KUKA KRL program: MyProgram_004().src

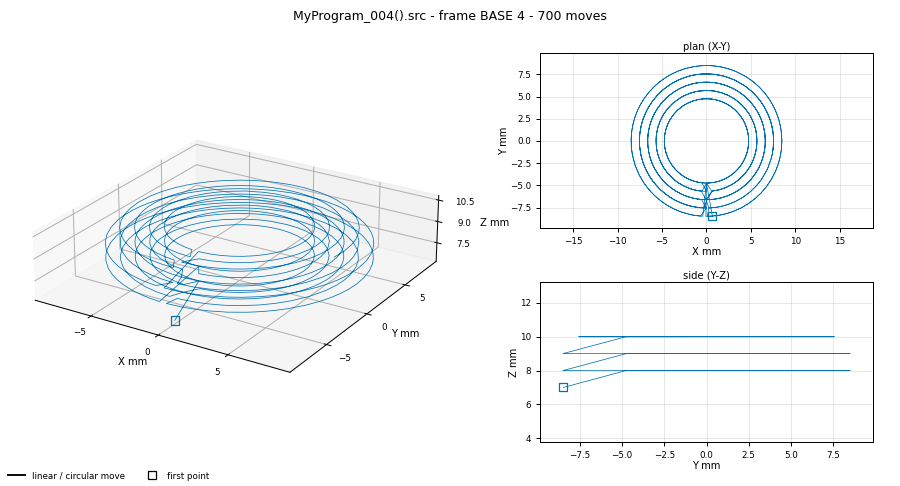
[picture p0: tool path of MyProgram_004().src in frame BASE 4, 700 of 700 moves have a stored position in this frame; points joined in program order, loops and branches not executed]
&ACCESS RVP
&REL 1
&PARAM TEMPLATE = C:\KRC\Roboter\Template\vorgabe
&PARAM EDITMASK = *
DEF MyProgram_004()
; ---- Setting reference (Base) ----
$BASE = BASE_DATA[4]

; --------------------------
; ---- Setting tool (TCP) ----
$TOOL = TOOL_DATA[3]
; --------------------------

$VEL.CP = VEL_APROX_PRINT
Startdeposition()
$VEL.CP = VEL_PRINT
LIN {X 0.6654,Y -8.462,Z 7,A -3.1447,B 0,C 0,E1 0.1598,E2 90.0714} C_DIS
Enddeposition()
LIN {X 0.0002,Y -4.7529,Z 8,A -2.9966,B 0,C 0,E1 0.1598,E2 90.0603} C_DIS
Startdeposition()
$VEL.CP = VEL_PRINT
LIN {X 0.0002,Y -4.7529,Z 8,A -3.0023,B 0,C 0,E1 0.1598,E2 90.066} C_DIS
LIN {X 0.816,Y -4.6799,Z 8,A -2.9741,B 0,C 0,E1 0.1598,E2 90.0709} C_DIS
LIN {X 1.4524,Y -4.5228,Z 8,A -2.9447,B 0,C 0,E1 0.1598,E2 90.0716} C_DIS
LIN {X 2.0618,Y -4.2811,Z 8,A -2.9121,B 0,C 0,E1 0.1598,E2 90.0716} C_DIS
LIN {X 2.6304,Y -3.9547,Z 8,A -2.8774,B 0,C 0,E1 0.1598,E2 90.0716} C_DIS
LIN {X 3.1509,Y -3.5562,Z 8,A -2.8413,B 0,C 0,E1 0.1598,E2 90.0717} C_DIS
LIN {X 3.6101,Y -3.0885,Z 8,A -2.8046,B 0,C 0,E1 0.1598,E2 90.0717} C_DIS
LIN {X 4.0002,Y -2.5617,Z 8,A -2.7679,B 0,C 0,E1 0.1598,E2 90.0717} C_DIS
LIN {X 4.3166,Y -1.9875,Z 8,A -2.7319,B 0,C 0,E1 0.1598,E2 90.0717} C_DIS
LIN {X 4.5475,Y -1.3739,Z 8,A -2.6974,B 0,C 0,E1 0.1598,E2 90.0717} C_DIS
LIN {X 4.6933,Y -0.7348,Z 8,A -2.6649,B 0,C 0,E1 0.1598,E2 90.0718} C_DIS
LIN {X 4.7495,Y -0.0819,Z 8,A -2.6352,B 0,C 0,E1 0.1598,E2 90.0718} C_DIS
LIN {X 4.7181,Y 0.573,Z 8,A -2.6086,B 0,C 0,E1 0.1598,E2 90.0718} C_DIS
LIN {X 4.5916,Y 1.2163,Z 8,A -2.586,B 0,C 0,E1 0.1598,E2 90.0718} C_DIS
LIN {X 4.3818,Y 1.8374,Z 8,A -2.5674,B 0,C 0,E1 0.1598,E2 90.0719} C_DIS
LIN {X 4.0877,Y 2.4234,Z 8,A -2.5534,B 0,C 0,E1 0.1598,E2 90.0719} C_DIS
LIN {X 3.7147,Y 2.9626,Z 8,A -2.5444,B 0,C 0,E1 0.1598,E2 90.072} C_DIS
LIN {X 3.2724,Y 3.4466,Z 8,A -2.5402,B 0,C 0,E1 0.1598,E2 90.072} C_DIS
LIN {X 2.7665,Y 3.864,Z 8,A -2.5413,B 0,C 0,E1 0.1598,E2 90.072} C_DIS
LIN {X 2.2075,Y 4.2066,Z 8,A -2.5474,B 0,C 0,E1 0.1598,E2 90.0721} C_DIS
LIN {X 1.6077,Y 4.4708,Z 8,A -2.5584,B 0,C 0,E1 0.1598,E2 90.0721} C_DIS
LIN {X 0.977,Y 4.6499,Z 8,A -2.5741,B 0,C 0,E1 0.1598,E2 90.0721} C_DIS
LIN {X 0.3277,Y 4.7412,Z 8,A -2.5942,B 0,C 0,E1 0.1598,E2 90.0721} C_DIS
LIN {X -0.3279,Y 4.7398,Z 8,A -2.6184,B 0,C 0,E1 0.1598,E2 90.0721} C_DIS
LIN {X -0.977,Y 4.6484,Z 8,A -2.6462,B 0,C 0,E1 0.1598,E2 90.0721} C_DIS
LIN {X -1.608,Y 4.4707,Z 8,A -2.677,B 0,C 0,E1 0.1598,E2 90.072} C_DIS
LIN {X -2.2078,Y 4.2061,Z 8,A -2.7102,B 0,C 0,E1 0.1598,E2 90.072} C_DIS
LIN {X -2.766,Y 3.862,Z 8,A -2.7453,B 0,C 0,E1 0.1598,E2 90.0719} C_DIS
LIN {X -3.2729,Y 3.4465,Z 8,A -2.7815,B 0,C 0,E1 0.1598,E2 90.0718} C_DIS
LIN {X -3.715,Y 2.9623,Z 8,A -2.8181,B 0,C 0,E1 0.1598,E2 90.0718} C_DIS
LIN {X -4.0878,Y 2.4229,Z 8,A -2.8545,B 0,C 0,E1 0.1598,E2 90.0716} C_DIS
LIN {X -4.3815,Y 1.8369,Z 8,A -2.89,B 0,C 0,E1 0.1598,E2 90.0716} C_DIS
LIN {X -4.5933,Y 1.2164,Z 8,A -2.924,B 0,C 0,E1 0.1598,E2 90.0715} C_DIS
LIN {X -4.7177,Y 0.5725,Z 8,A -2.9556,B 0,C 0,E1 0.1598,E2 90.0715} C_DIS
LIN {X -4.7506,Y -0.0822,Z 8,A -2.9844,B 0,C 0,E1 0.1598,E2 90.0714} C_DIS
LIN {X -4.6934,Y -0.7352,Z 8,A -3.0099,B 0,C 0,E1 0.1598,E2 90.0714} C_DIS
LIN {X -4.5474,Y -1.3743,Z 8,A -3.0314,B 0,C 0,E1 0.1598,E2 90.0714} C_DIS
LIN {X -4.3157,Y -1.9876,Z 8,A -3.0488,B 0,C 0,E1 0.1598,E2 90.0714} C_DIS
LIN {X -4.0017,Y -2.5632,Z 8,A -3.0616,B 0,C 0,E1 0.1598,E2 90.0714} C_DIS
LIN {X -3.6098,Y -3.0888,Z 8,A -3.0694,B 0,C 0,E1 0.1598,E2 90.0714} C_DIS
LIN {X -3.1503,Y -3.5561,Z 8,A -3.0722,B 0,C 0,E1 0.1598,E2 90.0714} C_DIS
LIN {X -2.6304,Y -3.9555,Z 8,A -3.0701,B 0,C 0,E1 0.1598,E2 90.0714} C_DIS
LIN {X -2.061,Y -4.2801,Z 8,A -3.0629,B 0,C 0,E1 0.1598,E2 90.0714} C_DIS
LIN {X -1.4527,Y -4.525,Z 8,A -3.0509,B 0,C 0,E1 0.1598,E2 90.0714} C_DIS
LIN {X -0.8159,Y -4.6817,Z 8,A -3.0342,B 0,C 0,E1 0.1598,E2 90.0715} C_DIS
LIN {X 0.0002,Y -4.7529,Z 8,A -3.0072,B 0,C 0,E1 0.1598,E2 90.0715} C_DIS
Enddeposition()
LIN {X 0.0002,Y -4.7529,Z 8,A -3.0072,B 0,C 0,E1 0.1598,E2 90.0715} C_DIS
Startdeposition()
$VEL.CP = VEL_PRINT
LIN {X -0.5157,Y -5.66,Z 8,A -3.0641,B 0,C 0,E1 0.1598,E2 90.0709} C_DIS
LIN {X -1.2329,Y -5.5494,Z 8,A -3.0863,B 0,C 0,E1 0.1598,E2 90.0714} C_DIS
LIN {X -2.1019,Y -5.2885,Z 8,A -3.1072,B 0,C 0,E1 0.1598,E2 90.0714} C_DIS
LIN {X -3.0914,Y -4.7699,Z 8,A -3.1214,B 0,C 0,E1 0.1598,E2 90.0712} C_DIS
LIN {X -3.7339,Y -4.2857,Z 8,A -3.1246,B 0,C 0,E1 0.1598,E2 90.0712} C_DIS
LIN {X -4.3031,Y -3.7167,Z 8,A -3.1215,B 0,C 0,E1 0.1598,E2 90.0712} C_DIS
LIN {X -4.784,Y -3.0715,Z 8,A -3.1119,B 0,C 0,E1 0.1598,E2 90.0712} C_DIS
LIN {X -5.0868,Y -2.5489,Z 8,A -3.101,B 0,C 0,E1 0.1598,E2 90.0713} C_DIS
LIN {X -5.4926,Y -1.467,Z 8,A -3.0698,B 0,C 0,E1 0.1598,E2 90.0708} C_DIS
LIN {X -5.6398,Y -0.761,Z 8,A -3.0457,B 0,C 0,E1 0.1598,E2 90.0711} C_DIS
LIN {X -5.6808,Y 0.176,Z 8,A -3.0077,B 0,C 0,E1 0.1598,E2 90.0711} C_DIS
LIN {X -5.6091,Y 0.9228,Z 8,A -2.9738,B 0,C 0,E1 0.1598,E2 90.0713} C_DIS
LIN {X -5.4394,Y 1.6537,Z 8,A -2.9367,B 0,C 0,E1 0.1598,E2 90.0713} C_DIS
LIN {X -5.1717,Y 2.3546,Z 8,A -2.8974,B 0,C 0,E1 0.1598,E2 90.0715} C_DIS
LIN {X -4.8184,Y 3.0165,Z 8,A -2.8565,B 0,C 0,E1 0.1598,E2 90.0715} C_DIS
LIN {X -4.3794,Y 3.6251,Z 8,A -2.8147,B 0,C 0,E1 0.1598,E2 90.0716} C_DIS
LIN {X -3.863,Y 4.1692,Z 8,A -2.7728,B 0,C 0,E1 0.1598,E2 90.0717} C_DIS
LIN {X -2.9369,Y 4.873,Z 8,A -2.7089,B 0,C 0,E1 0.1598,E2 90.0717} C_DIS
LIN {X -1.8956,Y 5.3645,Z 8,A -2.6499,B 0,C 0,E1 0.1598,E2 90.0719} C_DIS
LIN {X -1.0799,Y 5.5862,Z 8,A -2.6106,B 0,C 0,E1 0.1598,E2 90.0721} C_DIS
LIN {X 0.0829,Y 5.6834,Z 8,A -2.5636,B 0,C 0,E1 0.1598,E2 90.0721} C_DIS
LIN {X 0.8649,Y 5.6169,Z 8,A -2.5376,B 0,C 0,E1 0.1598,E2 90.0721} C_DIS
LIN {X 1.6302,Y 5.4433,Z 8,A -2.5166,B 0,C 0,E1 0.1598,E2 90.0721} C_DIS
LIN {X 2.3648,Y 5.1674,Z 8,A -2.5012,B 0,C 0,E1 0.1598,E2 90.0721} C_DIS
LIN {X 3.0553,Y 4.794,Z 8,A -2.4915,B 0,C 0,E1 0.1598,E2 90.0721} C_DIS
LIN {X 3.6858,Y 4.3265,Z 8,A -2.4879,B 0,C 0,E1 0.1598,E2 90.0721} C_DIS
LIN {X 4.2474,Y 3.7781,Z 8,A -2.4904,B 0,C 0,E1 0.1598,E2 90.0721} C_DIS
LIN {X 4.9144,Y 2.8699,Z 8,A -2.504,B 0,C 0,E1 0.1598,E2 90.0718} C_DIS
LIN {X 5.3537,Y 1.9124,Z 8,A -2.5283,B 0,C 0,E1 0.1598,E2 90.0718} C_DIS
LIN {X 5.5773,Y 1.1,Z 8,A -2.5546,B 0,C 0,E1 0.1598,E2 90.0718} C_DIS
LIN {X 5.6784,Y 0.2635,Z 8,A -2.5864,B 0,C 0,E1 0.1598,E2 90.0718} C_DIS
LIN {X 5.6566,Y -0.5791,Z 8,A -2.6229,B 0,C 0,E1 0.1598,E2 90.0717} C_DIS
LIN {X 5.5081,Y -1.4087,Z 8,A -2.6635,B 0,C 0,E1 0.1598,E2 90.0717} C_DIS
LIN {X 5.2396,Y -2.2076,Z 8,A -2.7073,B 0,C 0,E1 0.1598,E2 90.0717} C_DIS
LIN {X 4.9254,Y -2.8503,Z 8,A -2.7461,B 0,C 0,E1 0.1598,E2 90.0717} C_DIS
LIN {X 4.3094,Y -3.708,Z 8,A -2.8051,B 0,C 0,E1 0.1598,E2 90.0715} C_DIS
LIN {X 3.7119,Y -4.3055,Z 8,A -2.8525,B 0,C 0,E1 0.1598,E2 90.0715} C_DIS
LIN {X 3.0334,Y -4.8091,Z 8,A -2.8989,B 0,C 0,E1 0.1598,E2 90.0715} C_DIS
LIN {X 2.2871,Y -5.2051,Z 8,A -2.9431,B 0,C 0,E1 0.1598,E2 90.0715} C_DIS
LIN {X 1.4902,Y -5.4857,Z 8,A -2.9843,B 0,C 0,E1 0.1598,E2 90.0715} C_DIS
LIN {X 0.6608,Y -5.6458,Z 8,A -3.0215,B 0,C 0,E1 0.1598,E2 90.0715} C_DIS
LIN {X 0.6608,Y -5.6458,Z 8,A -3.0215,B 0,C 0,E1 0.1598,E2 90.0715} C_DIS
Enddeposition()
LIN {X 0.0648,Y -6.6225,Z 8,A -3.0837,B 0,C 0,E1 0.1598,E2 90.0703} C_DIS
Startdeposition()
$VEL.CP = VEL_PRINT
LIN {X 0.9354,Y -6.5522,Z 8,A -3.0499,B 0,C 0,E1 0.1598,E2 90.0714} C_DIS
LIN {X 1.6212,Y -6.4193,Z 8,A -3.0192,B 0,C 0,E1 0.1598,E2 90.0715} C_DIS
LIN {X 2.2882,Y -6.2108,Z 8,A -2.9859,B 0,C 0,E1 0.1598,E2 90.0715} C_DIS
LIN {X 2.9312,Y -5.9373,Z 8,A -2.9507,B 0,C 0,E1 0.1598,E2 90.0716} C_DIS
LIN {X 3.5398,Y -5.5941,Z 8,A -2.9137,B 0,C 0,E1 0.1598,E2 90.0716} C_DIS
LIN {X 4.1091,Y -5.1888,Z 8,A -2.8756,B 0,C 0,E1 0.1598,E2 90.0716} C_DIS
LIN {X 4.6332,Y -4.7267,Z 8,A -2.8368,B 0,C 0,E1 0.1598,E2 90.0716} C_DIS
LIN {X 5.1052,Y -4.2116,Z 8,A -2.7975,B 0,C 0,E1 0.1598,E2 90.0717} C_DIS
LIN {X 5.5227,Y -3.6513,Z 8,A -2.7584,B 0,C 0,E1 0.1598,E2 90.0717} C_DIS
LIN {X 5.8768,Y -3.0489,Z 8,A -2.7198,B 0,C 0,E1 0.1598,E2 90.0717} C_DIS
LIN {X 6.1649,Y -2.4124,Z 8,A -2.6822,B 0,C 0,E1 0.1598,E2 90.0717} C_DIS
LIN {X 6.3846,Y -1.7492,Z 8,A -2.6459,B 0,C 0,E1 0.1598,E2 90.0718} C_DIS
LIN {X 6.5333,Y -1.0664,Z 8,A -2.6115,B 0,C 0,E1 0.1598,E2 90.0718} C_DIS
LIN {X 6.6107,Y -0.372,Z 8,A -2.5792,B 0,C 0,E1 0.1598,E2 90.0718} C_DIS
LIN {X 6.6105,Y 0.3268,Z 8,A -2.5495,B 0,C 0,E1 0.1598,E2 90.0719} C_DIS
LIN {X 6.5388,Y 1.0217,Z 8,A -2.5227,B 0,C 0,E1 0.1598,E2 90.0719} C_DIS
LIN {X 6.3974,Y 1.706,Z 8,A -2.4989,B 0,C 0,E1 0.1598,E2 90.0719} C_DIS
LIN {X 6.1803,Y 2.3702,Z 8,A -2.4787,B 0,C 0,E1 0.1598,E2 90.072} C_DIS
LIN {X 5.8964,Y 3.0086,Z 8,A -2.4621,B 0,C 0,E1 0.1598,E2 90.072} C_DIS
LIN {X 5.5471,Y 3.6139,Z 8,A -2.4494,B 0,C 0,E1 0.1598,E2 90.072} C_DIS
LIN {X 5.1354,Y 4.1784,Z 8,A -2.4407,B 0,C 0,E1 0.1598,E2 90.0721} C_DIS
LIN {X 4.6656,Y 4.6955,Z 8,A -2.4361,B 0,C 0,E1 0.1598,E2 90.0721} C_DIS
LIN {X 4.1443,Y 5.1606,Z 8,A -2.4357,B 0,C 0,E1 0.1598,E2 90.0721} C_DIS
LIN {X 3.5773,Y 5.5689,Z 8,A -2.4394,B 0,C 0,E1 0.1598,E2 90.0722} C_DIS
LIN {X 2.9706,Y 5.9158,Z 8,A -2.4471,B 0,C 0,E1 0.1598,E2 90.0722} C_DIS
LIN {X 2.331,Y 6.1969,Z 8,A -2.4589,B 0,C 0,E1 0.1598,E2 90.0722} C_DIS
LIN {X 1.665,Y 6.4086,Z 8,A -2.4745,B 0,C 0,E1 0.1598,E2 90.0722} C_DIS
LIN {X 0.9803,Y 6.5482,Z 8,A -2.4939,B 0,C 0,E1 0.1598,E2 90.0722} C_DIS
LIN {X 0.2846,Y 6.6139,Z 8,A -2.5168,B 0,C 0,E1 0.1598,E2 90.0722} C_DIS
LIN {X -0.4142,Y 6.6069,Z 8,A -2.5429,B 0,C 0,E1 0.1598,E2 90.0722} C_DIS
LIN {X -1.1085,Y 6.5282,Z 8,A -2.5718,B 0,C 0,E1 0.1598,E2 90.0722} C_DIS
LIN {X -1.79,Y 6.3743,Z 8,A -2.6035,B 0,C 0,E1 0.1598,E2 90.0721} C_DIS
LIN {X -2.4518,Y 6.15,Z 8,A -2.6373,B 0,C 0,E1 0.1598,E2 90.0721} C_DIS
LIN {X -3.086,Y 5.8569,Z 8,A -2.6731,B 0,C 0,E1 0.1598,E2 90.072} C_DIS
LIN {X -3.6861,Y 5.4991,Z 8,A -2.7102,B 0,C 0,E1 0.1598,E2 90.0719} C_DIS
LIN {X -4.245,Y 5.0797,Z 8,A -2.7485,B 0,C 0,E1 0.1598,E2 90.0719} C_DIS
LIN {X -4.7551,Y 4.6024,Z 8,A -2.7874,B 0,C 0,E1 0.1598,E2 90.0717} C_DIS
LIN {X -5.2148,Y 4.0762,Z 8,A -2.8264,B 0,C 0,E1 0.1598,E2 90.0717} C_DIS
LIN {X -5.618,Y 3.5055,Z 8,A -2.8653,B 0,C 0,E1 0.1598,E2 90.0716} C_DIS
LIN {X -5.9566,Y 2.8942,Z 8,A -2.9035,B 0,C 0,E1 0.1598,E2 90.0716} C_DIS
LIN {X -6.2278,Y 2.2501,Z 8,A -2.9406,B 0,C 0,E1 0.1598,E2 90.0714} C_DIS
LIN {X -6.4294,Y 1.5809,Z 8,A -2.9761,B 0,C 0,E1 0.1598,E2 90.0714} C_DIS
LIN {X -6.5599,Y 0.8944,Z 8,A -3.0098,B 0,C 0,E1 0.1598,E2 90.0714} C_DIS
LIN {X -6.6156,Y 0.198,Z 8,A -3.0412,B 0,C 0,E1 0.1598,E2 90.0713} C_DIS
LIN {X -6.6007,Y -0.5005,Z 8,A -3.07,B 0,C 0,E1 0.1598,E2 90.0713} C_DIS
LIN {X -6.5106,Y -1.1935,Z 8,A -3.0959,B 0,C 0,E1 0.1598,E2 90.0713} C_DIS
LIN {X -6.3491,Y -1.8732,Z 8,A -3.1186,B 0,C 0,E1 0.1598,E2 90.0712} C_DIS
LIN {X -6.1165,Y -2.532,Z 8,A -3.1378,B 0,C 0,E1 0.1598,E2 90.0712} C_DIS
LIN {X -5.815,Y -3.1623,Z 8,A -3.1533,B 0,C 0,E1 0.1598,E2 90.0712} C_DIS
LIN {X -5.4482,Y -3.757,Z 8,A -3.165,B 0,C 0,E1 0.1598,E2 90.0712} C_DIS
LIN {X -5.0225,Y -4.3111,Z 8,A -3.1727,B 0,C 0,E1 0.1598,E2 90.0712} C_DIS
LIN {X -4.5415,Y -4.8179,Z 8,A -3.1765,B 0,C 0,E1 0.1598,E2 90.0712} C_DIS
LIN {X -4.0071,Y -5.2682,Z 8,A -3.1759,B 0,C 0,E1 0.1598,E2 90.0712} C_DIS
LIN {X -3.4299,Y -5.6621,Z 8,A -3.1714,B 0,C 0,E1 0.1598,E2 90.0712} C_DIS
LIN {X -2.8141,Y -5.9922,Z 8,A -3.1627,B 0,C 0,E1 0.1598,E2 90.0712} C_DIS
LIN {X -2.1668,Y -6.2556,Z 8,A -3.1501,B 0,C 0,E1 0.1598,E2 90.0713} C_DIS
LIN {X -1.4954,Y -6.4494,Z 8,A -3.1337,B 0,C 0,E1 0.1598,E2 90.0713} C_DIS
LIN {X -0.8068,Y -6.5688,Z 8,A -3.1135,B 0,C 0,E1 0.1598,E2 90.0714} C_DIS
LIN {X 0.0648,Y -6.6225,Z 8,A -3.0838,B 0,C 0,E1 0.1598,E2 90.0714} C_DIS
Enddeposition()
LIN {X 0.0648,Y -6.6225,Z 8,A -3.0838,B 0,C 0,E1 0.1598,E2 90.0714} C_DIS
Startdeposition()
$VEL.CP = VEL_PRINT
LIN {X -0.3005,Y -7.5521,Z 8,A -3.1362,B 0,C 0,E1 0.1598,E2 90.0708} C_DIS
LIN {X -1.3943,Y -7.4236,Z 8,A -3.1714,B 0,C 0,E1 0.1598,E2 90.0713} C_DIS
LIN {X -2.3277,Y -7.1896,Z 8,A -3.1957,B 0,C 0,E1 0.1598,E2 90.0713} C_DIS
LIN {X -3.4276,Y -6.7298,Z 8,A -3.2165,B 0,C 0,E1 0.1598,E2 90.0711} C_DIS
LIN {X -4.174,Y -6.2948,Z 8,A -3.2256,B 0,C 0,E1 0.1598,E2 90.0711} C_DIS
LIN {X -5.1254,Y -5.5535,Z 8,A -3.229,B 0,C 0,E1 0.1598,E2 90.071} C_DIS
LIN {X -5.9159,Y -4.6965,Z 8,A -3.2217,B 0,C 0,E1 0.1598,E2 90.0709} C_DIS
LIN {X -6.3665,Y -4.072,Z 8,A -3.212,B 0,C 0,E1 0.1598,E2 90.0709} C_DIS
LIN {X -6.9746,Y -2.9084,Z 8,A -3.1848,B 0,C 0,E1 0.1598,E2 90.0705} C_DIS
LIN {X -7.3445,Y -1.7591,Z 8,A -3.1501,B 0,C 0,E1 0.1598,E2 90.0706} C_DIS
LIN {X -7.5278,Y -0.6818,Z 8,A -3.1115,B 0,C 0,E1 0.1598,E2 90.0707} C_DIS
LIN {X -7.5337,Y 0.5991,Z 8,A -3.0576,B 0,C 0,E1 0.1598,E2 90.0705} C_DIS
LIN {X -7.3318,Y 1.8165,Z 8,A -2.999,B 0,C 0,E1 0.1598,E2 90.0707} C_DIS
LIN {X -7.098,Y 2.5925,Z 8,A -2.9581,B 0,C 0,E1 0.1598,E2 90.0712} C_DIS
LIN {X -6.64,Y 3.6072,Z 8,A -2.8985,B 0,C 0,E1 0.1598,E2 90.0712} C_DIS
LIN {X -6.088,Y 4.4712,Z 8,A -2.842,B 0,C 0,E1 0.1598,E2 90.0714} C_DIS
LIN {X -5.5672,Y 5.1049,Z 8,A -2.7962,B 0,C 0,E1 0.1598,E2 90.0716} C_DIS
LIN {X -4.8273,Y 5.8145,Z 8,A -2.739,B 0,C 0,E1 0.1598,E2 90.0716} C_DIS
LIN {X -3.9654,Y 6.4312,Z 8,A -2.6813,B 0,C 0,E1 0.1598,E2 90.0718} C_DIS
LIN {X -3.2143,Y 6.8395,Z 8,A -2.6365,B 0,C 0,E1 0.1598,E2 90.072} C_DIS
LIN {X -2.09,Y 7.2586,Z 8,A -2.5774,B 0,C 0,E1 0.1598,E2 90.072} C_DIS
LIN {X -1.381,Y 7.4314,Z 8,A -2.544,B 0,C 0,E1 0.1598,E2 90.0722} C_DIS
LIN {X -0.3666,Y 7.5493,Z 8,A -2.5016,B 0,C 0,E1 0.1598,E2 90.0722} C_DIS
LIN {X 0.952,Y 7.4973,Z 8,A -2.4551,B 0,C 0,E1 0.1598,E2 90.0722} C_DIS
LIN {X 2.1694,Y 7.2352,Z 8,A -2.4211,B 0,C 0,E1 0.1598,E2 90.0722} C_DIS
LIN {X 3.1883,Y 6.8521,Z 8,A -2.3996,B 0,C 0,E1 0.1598,E2 90.0722} C_DIS
LIN {X 4.2748,Y 6.2257,Z 8,A -2.3859,B 0,C 0,E1 0.1598,E2 90.0722} C_DIS
LIN {X 5.1495,Y 5.5305,Z 8,A -2.383,B 0,C 0,E1 0.1598,E2 90.0721} C_DIS
LIN {X 6.044,Y 4.5363,Z 8,A -2.3919,B 0,C 0,E1 0.1598,E2 90.0719} C_DIS
LIN {X 6.7773,Y 3.3424,Z 8,A -2.415,B 0,C 0,E1 0.1598,E2 90.0713} C_DIS
LIN {X 7.2345,Y 2.1842,Z 8,A -2.4475,B 0,C 0,E1 0.1598,E2 90.0716} C_DIS
LIN {X 7.4914,Y 0.9674,Z 8,A -2.4895,B 0,C 0,E1 0.1598,E2 90.0713} C_DIS
LIN {X 7.5545,Y 0.1953,Z 8,A -2.5203,B 0,C 0,E1 0.1598,E2 90.0717} C_DIS
LIN {X 7.5258,Y -0.7011,Z 8,A -2.5594,B 0,C 0,E1 0.1598,E2 90.0717} C_DIS
LIN {X 7.3499,Y -1.7618,Z 8,A -2.6108,B 0,C 0,E1 0.1598,E2 90.0715} C_DIS
LIN {X 6.9166,Y -3.0449,Z 8,A -2.681,B 0,C 0,E1 0.1598,E2 90.0712} C_DIS
LIN {X 6.2835,Y -4.1917,Z 8,A -2.7531,B 0,C 0,E1 0.1598,E2 90.0712} C_DIS
LIN {X 5.676,Y -4.9892,Z 8,A -2.8095,B 0,C 0,E1 0.1598,E2 90.0714} C_DIS
LIN {X 4.9446,Y -5.7142,Z 8,A -2.8672,B 0,C 0,E1 0.1598,E2 90.0714} C_DIS
LIN {X 3.9892,Y -6.4177,Z 8,A -2.9322,B 0,C 0,E1 0.1598,E2 90.0714} C_DIS
LIN {X 3.156,Y -6.8678,Z 8,A -2.982,B 0,C 0,E1 0.1598,E2 90.0715} C_DIS
LIN {X 2.1077,Y -7.2534,Z 8,A -3.0368,B 0,C 0,E1 0.1598,E2 90.0715} C_DIS
LIN {X 1.3502,Y -7.4321,Z 8,A -3.0722,B 0,C 0,E1 0.1598,E2 90.0715} C_DIS
LIN {X 0.2577,Y -7.5531,Z 8,A -3.1174,B 0,C 0,E1 0.1598,E2 90.0715} C_DIS
LIN {X 0.2577,Y -7.5531,Z 8,A -3.1174,B 0,C 0,E1 0.1598,E2 90.0715} C_DIS
Enddeposition()
LIN {X 0.0876,Y -8.49,Z 8,A -3.1623,B 0,C 0,E1 0.1598,E2 90.0702} C_DIS
Startdeposition()
$VEL.CP = VEL_PRINT
LIN {X 1.101,Y -8.4157,Z 8,A -3.1231,B 0,C 0,E1 0.1598,E2 90.0714} C_DIS
LIN {X 1.9012,Y -8.2718,Z 8,A -3.0878,B 0,C 0,E1 0.1598,E2 90.0714} C_DIS
LIN {X 2.877,Y -7.9881,Z 8,A -3.0399,B 0,C 0,E1 0.1598,E2 90.0714} C_DIS
LIN {X 3.8742,Y -7.5568,Z 8,A -2.985,B 0,C 0,E1 0.1598,E2 90.0715} C_DIS
LIN {X 4.8838,Y -6.9415,Z 8,A -2.9218,B 0,C 0,E1 0.1598,E2 90.0715} C_DIS
LIN {X 5.5503,Y -6.4222,Z 8,A -2.8753,B 0,C 0,E1 0.1598,E2 90.0716} C_DIS
LIN {X 6.1618,Y -5.8392,Z 8,A -2.8281,B 0,C 0,E1 0.1598,E2 90.0716} C_DIS
LIN {X 6.712,Y -5.1979,Z 8,A -2.7806,B 0,C 0,E1 0.1598,E2 90.0716} C_DIS
LIN {X 7.3552,Y -4.2442,Z 8,A -2.7163,B 0,C 0,E1 0.1598,E2 90.0716} C_DIS
LIN {X 7.824,Y -3.2899,Z 8,A -2.6585,B 0,C 0,E1 0.1598,E2 90.0716} C_DIS
LIN {X 8.1141,Y -2.4903,Z 8,A -2.614,B 0,C 0,E1 0.1598,E2 90.0717} C_DIS
LIN {X 8.3227,Y -1.6657,Z 8,A -2.5712,B 0,C 0,E1 0.1598,E2 90.0717} C_DIS
LIN {X 8.447,Y -0.8243,Z 8,A -2.5309,B 0,C 0,E1 0.1598,E2 90.0718} C_DIS
LIN {X 8.4862,Y 0.0253,Z 8,A -2.4934,B 0,C 0,E1 0.1598,E2 90.0718} C_DIS
LIN {X 8.4216,Y 1.0867,Z 8,A -2.4504,B 0,C 0,E1 0.1598,E2 90.0716} C_DIS
LIN {X 8.2013,Y 2.1972,Z 8,A -2.4114,B 0,C 0,E1 0.1598,E2 90.0716} C_DIS
LIN {X 7.8747,Y 3.1628,Z 8,A -2.3826,B 0,C 0,E1 0.1598,E2 90.0719} C_DIS
LIN {X 7.5351,Y 3.9043,Z 8,A -2.3638,B 0,C 0,E1 0.1598,E2 90.0721} C_DIS
LIN {X 7.126,Y 4.6099,Z 8,A -2.349,B 0,C 0,E1 0.1598,E2 90.0721} C_DIS
LIN {X 6.6513,Y 5.2731,Z 8,A -2.3385,B 0,C 0,E1 0.1598,E2 90.0721} C_DIS
LIN {X 5.974,Y 6.0351,Z 8,A -2.331,B 0,C 0,E1 0.1598,E2 90.0721} C_DIS
LIN {X 5.1729,Y 6.7304,Z 8,A -2.3313,B 0,C 0,E1 0.1598,E2 90.0721} C_DIS
LIN {X 4.4157,Y 7.2516,Z 8,A -2.3373,B 0,C 0,E1 0.1598,E2 90.0723} C_DIS
LIN {X 3.3989,Y 7.7782,Z 8,A -2.3526,B 0,C 0,E1 0.1598,E2 90.0723} C_DIS
LIN {X 2.6152,Y 8.0753,Z 8,A -2.3691,B 0,C 0,E1 0.1598,E2 90.0723} C_DIS
LIN {X 1.8062,Y 8.2944,Z 8,A -2.3897,B 0,C 0,E1 0.1598,E2 90.0723} C_DIS
LIN {X 0.9796,Y 8.4327,Z 8,A -2.4144,B 0,C 0,E1 0.1598,E2 90.0723} C_DIS
LIN {X 0.1434,Y 8.4878,Z 8,A -2.443,B 0,C 0,E1 0.1598,E2 90.0723} C_DIS
LIN {X -0.6942,Y 8.4592,Z 8,A -2.4751,B 0,C 0,E1 0.1598,E2 90.0723} C_DIS
LIN {X -1.5249,Y 8.3488,Z 8,A -2.5105,B 0,C 0,E1 0.1598,E2 90.0723} C_DIS
LIN {X -2.3408,Y 8.1575,Z 8,A -2.5487,B 0,C 0,E1 0.1598,E2 90.0722} C_DIS
LIN {X -3.1338,Y 7.8867,Z 8,A -2.5893,B 0,C 0,E1 0.1598,E2 90.0721} C_DIS
LIN {X -3.8964,Y 7.5392,Z 8,A -2.6321,B 0,C 0,E1 0.1598,E2 90.0721} C_DIS
LIN {X -4.621,Y 7.1183,Z 8,A -2.6765,B 0,C 0,E1 0.1598,E2 90.0719} C_DIS
LIN {X -5.3007,Y 6.6282,Z 8,A -2.7222,B 0,C 0,E1 0.1598,E2 90.0719} C_DIS
LIN {X -5.929,Y 6.0737,Z 8,A -2.7687,B 0,C 0,E1 0.1598,E2 90.0717} C_DIS
LIN {X -6.4992,Y 5.4597,Z 8,A -2.8155,B 0,C 0,E1 0.1598,E2 90.0717} C_DIS
LIN {X -7.0056,Y 4.792,Z 8,A -2.8622,B 0,C 0,E1 0.1598,E2 90.0715} C_DIS
LIN {X -7.4434,Y 4.0775,Z 8,A -2.9083,B 0,C 0,E1 0.1598,E2 90.0715} C_DIS
LIN {X -7.809,Y 3.3235,Z 8,A -2.9535,B 0,C 0,E1 0.1598,E2 90.0714} C_DIS
LIN {X -8.0987,Y 2.5372,Z 8,A -2.9972,B 0,C 0,E1 0.1598,E2 90.0713} C_DIS
LIN {X -8.3099,Y 1.7263,Z 8,A -3.039,B 0,C 0,E1 0.1598,E2 90.0712} C_DIS
LIN {X -8.4401,Y 0.8986,Z 8,A -3.0786,B 0,C 0,E1 0.1598,E2 90.0712} C_DIS
LIN {X -8.4875,Y 0.0619,Z 8,A -3.1155,B 0,C 0,E1 0.1598,E2 90.0711} C_DIS
LIN {X -8.4507,Y -0.7752,Z 8,A -3.1494,B 0,C 0,E1 0.1598,E2 90.0711} C_DIS
LIN {X -8.3333,Y -1.6049,Z 8,A -3.18,B 0,C 0,E1 0.1598,E2 90.071} C_DIS
LIN {X -8.018,Y -2.7956,Z 8,A -3.2182,B 0,C 0,E1 0.1598,E2 90.0706} C_DIS
LIN {X -7.5653,Y -3.8469,Z 8,A -3.2459,B 0,C 0,E1 0.1598,E2 90.0706} C_DIS
LIN {X -7.1388,Y -4.5901,Z 8,A -3.2618,B 0,C 0,E1 0.1598,E2 90.0709} C_DIS
LIN {X -6.6397,Y -5.2866,Z 8,A -3.2729,B 0,C 0,E1 0.1598,E2 90.0709} C_DIS
LIN {X -5.851,Y -6.1519,Z 8,A -3.2804,B 0,C 0,E1 0.1598,E2 90.0709} C_DIS
LIN {X -5.0988,Y -6.7842,Z 8,A -3.2796,B 0,C 0,E1 0.1598,E2 90.071} C_DIS
LIN {X -4.4501,Y -7.228,Z 8,A -3.2746,B 0,C 0,E1 0.1598,E2 90.071} C_DIS
LIN {X -3.5864,Y -7.6966,Z 8,A -3.2627,B 0,C 0,E1 0.1598,E2 90.071} C_DIS
LIN {X -2.8051,Y -8.0145,Z 8,A -3.2476,B 0,C 0,E1 0.1598,E2 90.0712} C_DIS
LIN {X -1.7581,Y -8.3051,Z 8,A -3.2215,B 0,C 0,E1 0.1598,E2 90.0712} C_DIS
LIN {X -1.0919,Y -8.4178,Z 8,A -3.2019,B 0,C 0,E1 0.1598,E2 90.0712} C_DIS
LIN {X -0.419,Y -8.4781,Z 8,A -3.1798,B 0,C 0,E1 0.1598,E2 90.0713} C_DIS
LIN {X -0.419,Y -8.4781,Z 8,A -3.1798,B 0,C 0,E1 0.1598,E2 90.0713} C_DIS
Enddeposition()
LIN {X 0.0002,Y -4.753,Z 9,A -2.9914,B 0,C 0,E1 0.1598,E2 90.0603} C_DIS
Startdeposition()
$VEL.CP = VEL_PRINT
LIN {X 0.0002,Y -4.753,Z 9,A -2.997,B 0,C 0,E1 0.1598,E2 90.066} C_DIS
LIN {X -0.816,Y -4.6818,Z 9,A -3.0288,B 0,C 0,E1 0.1598,E2 90.0709} C_DIS
LIN {X -1.4526,Y -4.5248,Z 9,A -3.0462,B 0,C 0,E1 0.1598,E2 90.0715} C_DIS
LIN {X -2.061,Y -4.2801,Z 9,A -3.0582,B 0,C 0,E1 0.1598,E2 90.0715} C_DIS
LIN {X -2.6305,Y -3.9555,Z 9,A -3.0654,B 0,C 0,E1 0.1598,E2 90.0715} C_DIS
LIN {X -3.1503,Y -3.5561,Z 9,A -3.0676,B 0,C 0,E1 0.1598,E2 90.0714} C_DIS
LIN {X -3.6097,Y -3.0887,Z 9,A -3.0647,B 0,C 0,E1 0.1598,E2 90.0714} C_DIS
LIN {X -4.0017,Y -2.5631,Z 9,A -3.0569,B 0,C 0,E1 0.1598,E2 90.0714} C_DIS
LIN {X -4.3158,Y -1.9876,Z 9,A -3.0441,B 0,C 0,E1 0.1598,E2 90.0714} C_DIS
LIN {X -4.5474,Y -1.3743,Z 9,A -3.0267,B 0,C 0,E1 0.1598,E2 90.0714} C_DIS
LIN {X -4.6934,Y -0.7352,Z 9,A -3.0051,B 0,C 0,E1 0.1598,E2 90.0714} C_DIS
LIN {X -4.7505,Y -0.0822,Z 9,A -2.9797,B 0,C 0,E1 0.1598,E2 90.0714} C_DIS
LIN {X -4.7177,Y 0.5725,Z 9,A -2.9509,B 0,C 0,E1 0.1598,E2 90.0714} C_DIS
LIN {X -4.5934,Y 1.2165,Z 9,A -2.9192,B 0,C 0,E1 0.1598,E2 90.0714} C_DIS
LIN {X -4.3816,Y 1.837,Z 9,A -2.8852,B 0,C 0,E1 0.1598,E2 90.0715} C_DIS
LIN {X -4.0872,Y 2.4226,Z 9,A -2.8497,B 0,C 0,E1 0.1598,E2 90.0716} C_DIS
LIN {X -3.7154,Y 2.9626,Z 9,A -2.8133,B 0,C 0,E1 0.1598,E2 90.0716} C_DIS
LIN {X -3.2729,Y 3.4465,Z 9,A -2.7766,B 0,C 0,E1 0.1598,E2 90.0718} C_DIS
LIN {X -2.7656,Y 3.8617,Z 9,A -2.7404,B 0,C 0,E1 0.1598,E2 90.0718} C_DIS
LIN {X -2.2086,Y 4.2074,Z 9,A -2.7053,B 0,C 0,E1 0.1598,E2 90.0719} C_DIS
LIN {X -1.6086,Y 4.4721,Z 9,A -2.6721,B 0,C 0,E1 0.1598,E2 90.0719} C_DIS
LIN {X -0.977,Y 4.6483,Z 9,A -2.6414,B 0,C 0,E1 0.1598,E2 90.072} C_DIS
LIN {X -0.328,Y 4.7397,Z 9,A -2.6136,B 0,C 0,E1 0.1598,E2 90.072} C_DIS
LIN {X 0.3276,Y 4.7413,Z 9,A -2.5894,B 0,C 0,E1 0.1598,E2 90.0721} C_DIS
LIN {X 0.9769,Y 4.6499,Z 9,A -2.5693,B 0,C 0,E1 0.1598,E2 90.0721} C_DIS
LIN {X 1.6076,Y 4.4709,Z 9,A -2.5536,B 0,C 0,E1 0.1598,E2 90.0721} C_DIS
LIN {X 2.2074,Y 4.2067,Z 9,A -2.5426,B 0,C 0,E1 0.1598,E2 90.0721} C_DIS
LIN {X 2.7665,Y 3.864,Z 9,A -2.5365,B 0,C 0,E1 0.1598,E2 90.0721} C_DIS
LIN {X 3.2723,Y 3.4467,Z 9,A -2.5354,B 0,C 0,E1 0.1598,E2 90.0721} C_DIS
LIN {X 3.7147,Y 2.9627,Z 9,A -2.5396,B 0,C 0,E1 0.1598,E2 90.0721} C_DIS
LIN {X 4.0878,Y 2.4236,Z 9,A -2.5486,B 0,C 0,E1 0.1598,E2 90.0721} C_DIS
LIN {X 4.3811,Y 1.8372,Z 9,A -2.5626,B 0,C 0,E1 0.1598,E2 90.072} C_DIS
LIN {X 4.5923,Y 1.2166,Z 9,A -2.5811,B 0,C 0,E1 0.1598,E2 90.072} C_DIS
LIN {X 4.7181,Y 0.5731,Z 9,A -2.6037,B 0,C 0,E1 0.1598,E2 90.0719} C_DIS
LIN {X 4.7496,Y -0.0818,Z 9,A -2.6303,B 0,C 0,E1 0.1598,E2 90.0719} C_DIS
LIN {X 4.6933,Y -0.7347,Z 9,A -2.6601,B 0,C 0,E1 0.1598,E2 90.0718} C_DIS
LIN {X 4.5491,Y -1.3743,Z 9,A -2.6925,B 0,C 0,E1 0.1598,E2 90.0718} C_DIS
LIN {X 4.3154,Y -1.9869,Z 9,A -2.7271,B 0,C 0,E1 0.1598,E2 90.0718} C_DIS
LIN {X 4.0002,Y -2.5616,Z 9,A -2.7631,B 0,C 0,E1 0.1598,E2 90.0718} C_DIS
LIN {X 3.6102,Y -3.0884,Z 9,A -2.7998,B 0,C 0,E1 0.1598,E2 90.0718} C_DIS
LIN {X 3.1508,Y -3.556,Z 9,A -2.8365,B 0,C 0,E1 0.1598,E2 90.0717} C_DIS
LIN {X 2.6305,Y -3.9547,Z 9,A -2.8725,B 0,C 0,E1 0.1598,E2 90.0717} C_DIS
LIN {X 2.0617,Y -4.2807,Z 9,A -2.9072,B 0,C 0,E1 0.1598,E2 90.0717} C_DIS
LIN {X 1.374,Y -4.5466,Z 9,A -2.9438,B 0,C 0,E1 0.1598,E2 90.0717} C_DIS
LIN {X 0.8161,Y -4.6803,Z 9,A -2.9699,B 0,C 0,E1 0.1598,E2 90.0717} C_DIS
LIN {X 0.0002,Y -4.753,Z 9,A -3.003,B 0,C 0,E1 0.1598,E2 90.0716} C_DIS
Enddeposition()
LIN {X 0.0002,Y -4.753,Z 9,A -3.003,B 0,C 0,E1 0.1598,E2 90.0716} C_DIS
Startdeposition()
$VEL.CP = VEL_PRINT
LIN {X 0.5909,Y -5.6516,Z 9,A -3.0189,B 0,C 0,E1 0.1598,E2 90.071} C_DIS
LIN {X 1.374,Y -5.5148,Z 9,A -2.9849,B 0,C 0,E1 0.1598,E2 90.0716} C_DIS
LIN {X 2.1302,Y -5.2694,Z 9,A -2.9467,B 0,C 0,E1 0.1598,E2 90.0716} C_DIS
LIN {X 2.8452,Y -4.9214,Z 9,A -2.9057,B 0,C 0,E1 0.1598,E2 90.0716} C_DIS
LIN {X 3.5045,Y -4.4764,Z 9,A -2.8626,B 0,C 0,E1 0.1598,E2 90.0716} C_DIS
LIN {X 4.0948,Y -3.9434,Z 9,A -2.8183,B 0,C 0,E1 0.1598,E2 90.0716} C_DIS
LIN {X 4.6044,Y -3.3327,Z 9,A -2.7736,B 0,C 0,E1 0.1598,E2 90.0716} C_DIS
LIN {X 5.0254,Y -2.6582,Z 9,A -2.7295,B 0,C 0,E1 0.1598,E2 90.0716} C_DIS
LIN {X 5.3452,Y -1.9301,Z 9,A -2.6868,B 0,C 0,E1 0.1598,E2 90.0717} C_DIS
LIN {X 5.5628,Y -1.1654,Z 9,A -2.6463,B 0,C 0,E1 0.1598,E2 90.0717} C_DIS
LIN {X 5.6703,Y -0.3776,Z 9,A -2.6089,B 0,C 0,E1 0.1598,E2 90.0717} C_DIS
LIN {X 5.6676,Y 0.4173,Z 9,A -2.5753,B 0,C 0,E1 0.1598,E2 90.0717} C_DIS
LIN {X 5.5536,Y 1.2041,Z 9,A -2.5461,B 0,C 0,E1 0.1598,E2 90.0718} C_DIS
LIN {X 5.3326,Y 1.9678,Z 9,A -2.5219,B 0,C 0,E1 0.1598,E2 90.0718} C_DIS
LIN {X 4.9144,Y 2.8698,Z 9,A -2.4989,B 0,C 0,E1 0.1598,E2 90.0718} C_DIS
LIN {X 4.2487,Y 3.7767,Z 9,A -2.4851,B 0,C 0,E1 0.1598,E2 90.0718} C_DIS
LIN {X 3.689,Y 4.3237,Z 9,A -2.4828,B 0,C 0,E1 0.1598,E2 90.0721} C_DIS
LIN {X 3.0607,Y 4.7903,Z 9,A -2.4863,B 0,C 0,E1 0.1598,E2 90.0721} C_DIS
LIN {X 2.3729,Y 5.1636,Z 9,A -2.496,B 0,C 0,E1 0.1598,E2 90.0721} C_DIS
LIN {X 1.641,Y 5.4399,Z 9,A -2.5113,B 0,C 0,E1 0.1598,E2 90.0721} C_DIS
LIN {X 0.8785,Y 5.6158,Z 9,A -2.532,B 0,C 0,E1 0.1598,E2 90.0721} C_DIS
LIN {X 0.0988,Y 5.6842,Z 9,A -2.5579,B 0,C 0,E1 0.1598,E2 90.0721} C_DIS
LIN {X -1.0646,Y 5.5892,Z 9,A -2.6048,B 0,C 0,E1 0.1598,E2 90.0721} C_DIS
LIN {X -1.8585,Y 5.378,Z 9,A -2.643,B 0,C 0,E1 0.1598,E2 90.0721} C_DIS
LIN {X -2.6452,Y 5.0381,Z 9,A -2.6863,B 0,C 0,E1 0.1598,E2 90.0719} C_DIS
LIN {X -3.7683,Y 4.2632,Z 9,A -2.7602,B 0,C 0,E1 0.1598,E2 90.0716} C_DIS
LIN {X -4.4145,Y 3.579,Z 9,A -2.8129,B 0,C 0,E1 0.1598,E2 90.0716} C_DIS
LIN {X -4.8501,Y 2.9648,Z 9,A -2.8548,B 0,C 0,E1 0.1598,E2 90.0716} C_DIS
LIN {X -5.1985,Y 2.2974,Z 9,A -2.8957,B 0,C 0,E1 0.1598,E2 90.0715} C_DIS
LIN {X -5.4592,Y 1.5909,Z 9,A -2.9351,B 0,C 0,E1 0.1598,E2 90.0715} C_DIS
LIN {X -5.6667,Y 0.5072,Z 9,A -2.988,B 0,C 0,E1 0.1598,E2 90.071} C_DIS
LIN {X -5.6437,Y -0.7264,Z 9,A -3.039,B 0,C 0,E1 0.1598,E2 90.0708} C_DIS
LIN {X -5.4991,Y -1.4412,Z 9,A -3.0643,B 0,C 0,E1 0.1598,E2 90.0712} C_DIS
LIN {X -5.292,Y -2.0936,Z 9,A -3.0842,B 0,C 0,E1 0.1598,E2 90.0712} C_DIS
LIN {X -4.9859,Y -2.7331,Z 9,A -3.0999,B 0,C 0,E1 0.1598,E2 90.0712} C_DIS
LIN {X -4.5322,Y -3.4316,Z 9,A -3.1127,B 0,C 0,E1 0.1598,E2 90.0712} C_DIS
LIN {X -3.9815,Y -4.0562,Z 9,A -3.1189,B 0,C 0,E1 0.1598,E2 90.0712} C_DIS
LIN {X -3.3468,Y -4.5956,Z 9,A -3.1184,B 0,C 0,E1 0.1598,E2 90.0712} C_DIS
LIN {X -2.6388,Y -5.034,Z 9,A -3.111,B 0,C 0,E1 0.1598,E2 90.0713} C_DIS
LIN {X -1.5416,Y -5.4778,Z 9,A -3.0894,B 0,C 0,E1 0.1598,E2 90.0713} C_DIS
LIN {X -0.5865,Y -5.6532,Z 9,A -3.0619,B 0,C 0,E1 0.1598,E2 90.0715} C_DIS
LIN {X -0.5865,Y -5.6532,Z 9,A -3.0619,B 0,C 0,E1 0.1598,E2 90.0715} C_DIS
Enddeposition()
LIN {X -0.0377,Y -6.6237,Z 9,A -3.0819,B 0,C 0,E1 0.1598,E2 90.0703} C_DIS
Startdeposition()
$VEL.CP = VEL_PRINT
LIN {X -0.9084,Y -6.5552,Z 9,A -3.112,B 0,C 0,E1 0.1598,E2 90.0714} C_DIS
LIN {X -1.5947,Y -6.424,Z 9,A -3.1317,B 0,C 0,E1 0.1598,E2 90.0714} C_DIS
LIN {X -2.2636,Y -6.2219,Z 9,A -3.1476,B 0,C 0,E1 0.1598,E2 90.0714} C_DIS
LIN {X -2.9066,Y -5.9484,Z 9,A -3.1597,B 0,C 0,E1 0.1598,E2 90.0714} C_DIS
LIN {X -3.5162,Y -5.6067,Z 9,A -3.1676,B 0,C 0,E1 0.1598,E2 90.0713} C_DIS
LIN {X -4.0876,Y -5.2048,Z 9,A -3.1715,B 0,C 0,E1 0.1598,E2 90.0713} C_DIS
LIN {X -4.6144,Y -4.7459,Z 9,A -3.1715,B 0,C 0,E1 0.1598,E2 90.0713} C_DIS
LIN {X -5.0889,Y -4.2329,Z 9,A -3.1672,B 0,C 0,E1 0.1598,E2 90.0713} C_DIS
LIN {X -5.5062,Y -3.6725,Z 9,A -3.1589,B 0,C 0,E1 0.1598,E2 90.0712} C_DIS
LIN {X -5.863,Y -3.0718,Z 9,A -3.1466,B 0,C 0,E1 0.1598,E2 90.0712} C_DIS
LIN {X -6.1549,Y -2.437,Z 9,A -3.1306,B 0,C 0,E1 0.1598,E2 90.0712} C_DIS
LIN {X -6.378,Y -1.7748,Z 9,A -3.1108,B 0,C 0,E1 0.1598,E2 90.0712} C_DIS
LIN {X -6.5272,Y -1.0923,Z 9,A -3.0876,B 0,C 0,E1 0.1598,E2 90.0712} C_DIS
LIN {X -6.6085,Y -0.3984,Z 9,A -3.0613,B 0,C 0,E1 0.1598,E2 90.0712} C_DIS
LIN {X -6.6127,Y 0.3004,Z 9,A -3.032,B 0,C 0,E1 0.1598,E2 90.0712} C_DIS
LIN {X -6.546,Y 0.9959,Z 9,A -3.0003,B 0,C 0,E1 0.1598,E2 90.0713} C_DIS
LIN {X -6.4037,Y 1.6801,Z 9,A -2.9663,B 0,C 0,E1 0.1598,E2 90.0713} C_DIS
LIN {X -6.191,Y 2.3457,Z 9,A -2.9304,B 0,C 0,E1 0.1598,E2 90.0714} C_DIS
LIN {X -5.9097,Y 2.9852,Z 9,A -2.8931,B 0,C 0,E1 0.1598,E2 90.0715} C_DIS
LIN {X -5.5617,Y 3.5911,Z 9,A -2.8548,B 0,C 0,E1 0.1598,E2 90.0715} C_DIS
LIN {X -5.1517,Y 4.157,Z 9,A -2.8159,B 0,C 0,E1 0.1598,E2 90.0717} C_DIS
LIN {X -4.6844,Y 4.6765,Z 9,A -2.7768,B 0,C 0,E1 0.1598,E2 90.0717} C_DIS
LIN {X -4.1662,Y 5.145,Z 9,A -2.738,B 0,C 0,E1 0.1598,E2 90.0718} C_DIS
LIN {X -3.6006,Y 5.5555,Z 9,A -2.6999,B 0,C 0,E1 0.1598,E2 90.0718} C_DIS
LIN {X -2.9948,Y 5.9038,Z 9,A -2.6629,B 0,C 0,E1 0.1598,E2 90.072} C_DIS
LIN {X -2.3564,Y 6.1877,Z 9,A -2.6274,B 0,C 0,E1 0.1598,E2 90.072} C_DIS
LIN {X -1.6914,Y 6.4025,Z 9,A -2.5938,B 0,C 0,E1 0.1598,E2 90.072} C_DIS
LIN {X -1.0073,Y 6.5448,Z 9,A -2.5626,B 0,C 0,E1 0.1598,E2 90.0721} C_DIS
LIN {X -0.3118,Y 6.6116,Z 9,A -2.5341,B 0,C 0,E1 0.1598,E2 90.0721} C_DIS
LIN {X 0.3869,Y 6.6076,Z 9,A -2.5085,B 0,C 0,E1 0.1598,E2 90.0722} C_DIS
LIN {X 1.0814,Y 6.5313,Z 9,A -2.4861,B 0,C 0,E1 0.1598,E2 90.0722} C_DIS
LIN {X 1.7638,Y 6.3811,Z 9,A -2.4672,B 0,C 0,E1 0.1598,E2 90.0722} C_DIS
LIN {X 2.4264,Y 6.1593,Z 9,A -2.4521,B 0,C 0,E1 0.1598,E2 90.0722} C_DIS
LIN {X 3.0614,Y 5.8679,Z 9,A -2.441,B 0,C 0,E1 0.1598,E2 90.0722} C_DIS
LIN {X 3.6636,Y 5.5136,Z 9,A -2.4337,B 0,C 0,E1 0.1598,E2 90.0722} C_DIS
LIN {X 4.2247,Y 5.097,Z 9,A -2.4307,B 0,C 0,E1 0.1598,E2 90.0722} C_DIS
LIN {X 4.7386,Y 4.6235,Z 9,A -2.4317,B 0,C 0,E1 0.1598,E2 90.0722} C_DIS
LIN {X 5.2,Y 4.0988,Z 9,A -2.4369,B 0,C 0,E1 0.1598,E2 90.0722} C_DIS
LIN {X 5.6021,Y 3.5273,Z 9,A -2.4462,B 0,C 0,E1 0.1598,E2 90.0722} C_DIS
LIN {X 5.9435,Y 2.9175,Z 9,A -2.4595,B 0,C 0,E1 0.1598,E2 90.0721} C_DIS
LIN {X 6.216,Y 2.2741,Z 9,A -2.4767,B 0,C 0,E1 0.1598,E2 90.0721} C_DIS
LIN {X 6.421,Y 1.6062,Z 9,A -2.4974,B 0,C 0,E1 0.1598,E2 90.072} C_DIS
LIN {X 6.5557,Y 0.9205,Z 9,A -2.5216,B 0,C 0,E1 0.1598,E2 90.072} C_DIS
LIN {X 6.6138,Y 0.2242,Z 9,A -2.5489,B 0,C 0,E1 0.1598,E2 90.072} C_DIS
LIN {X 6.6035,Y -0.4744,Z 9,A -2.579,B 0,C 0,E1 0.1598,E2 90.0719} C_DIS
LIN {X 6.5158,Y -1.1675,Z 9,A -2.6116,B 0,C 0,E1 0.1598,E2 90.0719} C_DIS
LIN {X 6.357,Y -1.848,Z 9,A -2.6463,B 0,C 0,E1 0.1598,E2 90.0718} C_DIS
LIN {X 6.1274,Y -2.5079,Z 9,A -2.6828,B 0,C 0,E1 0.1598,E2 90.0718} C_DIS
LIN {X 5.8296,Y -3.14,Z 9,A -2.7206,B 0,C 0,E1 0.1598,E2 90.0718} C_DIS
LIN {X 5.4653,Y -3.7362,Z 9,A -2.7593,B 0,C 0,E1 0.1598,E2 90.0718} C_DIS
LIN {X 5.0394,Y -4.2902,Z 9,A -2.7985,B 0,C 0,E1 0.1598,E2 90.0717} C_DIS
LIN {X 4.559,Y -4.7975,Z 9,A -2.8377,B 0,C 0,E1 0.1598,E2 90.0717} C_DIS
LIN {X 4.0279,Y -5.2515,Z 9,A -2.8764,B 0,C 0,E1 0.1598,E2 90.0717} C_DIS
LIN {X 3.4526,Y -5.6481,Z 9,A -2.9144,B 0,C 0,E1 0.1598,E2 90.0717} C_DIS
LIN {X 2.8386,Y -5.9813,Z 9,A -2.9511,B 0,C 0,E1 0.1598,E2 90.0716} C_DIS
LIN {X 2.1917,Y -6.2455,Z 9,A -2.986,B 0,C 0,E1 0.1598,E2 90.0716} C_DIS
LIN {X 1.5214,Y -6.4428,Z 9,A -3.019,B 0,C 0,E1 0.1598,E2 90.0716} C_DIS
LIN {X 0.8338,Y -6.5662,Z 9,A -3.0495,B 0,C 0,E1 0.1598,E2 90.0716} C_DIS
LIN {X -0.0377,Y -6.6237,Z 9,A -3.0839,B 0,C 0,E1 0.1598,E2 90.0715} C_DIS
Enddeposition()
LIN {X -0.0377,Y -6.6237,Z 9,A -3.0839,B 0,C 0,E1 0.1598,E2 90.0715} C_DIS
Startdeposition()
$VEL.CP = VEL_PRINT
LIN {X 0.2712,Y -7.5528,Z 9,A -3.1115,B 0,C 0,E1 0.1598,E2 90.0709} C_DIS
LIN {X 1.3609,Y -7.435,Z 9,A -3.0671,B 0,C 0,E1 0.1598,E2 90.0715} C_DIS
LIN {X 2.3592,Y -7.1742,Z 9,A -3.0194,B 0,C 0,E1 0.1598,E2 90.0715} C_DIS
LIN {X 3.128,Y -6.8739,Z 9,A -2.9785,B 0,C 0,E1 0.1598,E2 90.0715} C_DIS
LIN {X 4.1281,Y -6.3317,Z 9,A -2.9187,B 0,C 0,E1 0.1598,E2 90.0715} C_DIS
LIN {X 4.8588,Y -5.7876,Z 9,A -2.8688,B 0,C 0,E1 0.1598,E2 90.0715} C_DIS
LIN {X 5.6081,Y -5.0597,Z 9,A -2.8103,B 0,C 0,E1 0.1598,E2 90.0715} C_DIS
LIN {X 6.1325,Y -4.4089,Z 9,A -2.7634,B 0,C 0,E1 0.1598,E2 90.0717} C_DIS
LIN {X 6.8293,Y -3.2353,Z 9,A -2.6874,B 0,C 0,E1 0.1598,E2 90.0712} C_DIS
LIN {X 7.2523,Y -2.1103,Z 9,A -2.6242,B 0,C 0,E1 0.1598,E2 90.0714} C_DIS
LIN {X 7.4577,Y -1.2196,Z 9,A -2.579,B 0,C 0,E1 0.1598,E2 90.0716} C_DIS
LIN {X 7.5546,Y -0.188,Z 9,A -2.5315,B 0,C 0,E1 0.1598,E2 90.0716} C_DIS
LIN {X 7.5238,Y 0.7187,Z 9,A -2.4943,B 0,C 0,E1 0.1598,E2 90.0717} C_DIS
LIN {X 7.3888,Y 1.5847,Z 9,A -2.4626,B 0,C 0,E1 0.1598,E2 90.0719} C_DIS
LIN {X 7.1039,Y 2.5763,Z 9,A -2.4309,B 0,C 0,E1 0.1598,E2 90.0718} C_DIS
LIN {X 6.4886,Y 3.8745,Z 9,A -2.3981,B 0,C 0,E1 0.1598,E2 90.0715} C_DIS
LIN {X 5.893,Y 4.7244,Z 9,A -2.3845,B 0,C 0,E1 0.1598,E2 90.072} C_DIS
LIN {X 5.1922,Y 5.49,Z 9,A -2.378,B 0,C 0,E1 0.1598,E2 90.072} C_DIS
LIN {X 4.345,Y 6.1767,Z 9,A -2.3803,B 0,C 0,E1 0.1598,E2 90.0721} C_DIS
LIN {X 3.1904,Y 6.8511,Z 9,A -2.3943,B 0,C 0,E1 0.1598,E2 90.0721} C_DIS
LIN {X 1.95,Y 7.3009,Z 9,A -2.4213,B 0,C 0,E1 0.1598,E2 90.0722} C_DIS
LIN {X 0.8244,Y 7.5086,Z 9,A -2.4542,B 0,C 0,E1 0.1598,E2 90.0722} C_DIS
LIN {X -0.3793,Y 7.5485,Z 9,A -2.497,B 0,C 0,E1 0.1598,E2 90.0722} C_DIS
LIN {X -1.36,Y 7.4351,Z 9,A -2.5379,B 0,C 0,E1 0.1598,E2 90.0722} C_DIS
LIN {X -2.2381,Y 7.2176,Z 9,A -2.5795,B 0,C 0,E1 0.1598,E2 90.0722} C_DIS
LIN {X -3.187,Y 6.8527,Z 9,A -2.6299,B 0,C 0,E1 0.1598,E2 90.072} C_DIS
LIN {X -3.9539,Y 6.4388,Z 9,A -2.6756,B 0,C 0,E1 0.1598,E2 90.072} C_DIS
LIN {X -4.6695,Y 5.9414,Z 9,A -2.7229,B 0,C 0,E1 0.1598,E2 90.0718} C_DIS
LIN {X -5.2983,Y 5.3893,Z 9,A -2.7693,B 0,C 0,E1 0.1598,E2 90.0718} C_DIS
LIN {X -6.0887,Y 4.4686,Z 9,A -2.8369,B 0,C 0,E1 0.1598,E2 90.0713} C_DIS
LIN {X -6.7369,Y 3.4256,Z 9,A -2.9046,B 0,C 0,E1 0.1598,E2 90.0712} C_DIS
LIN {X -7.1578,Y 2.4105,Z 9,A -2.9628,B 0,C 0,E1 0.1598,E2 90.0712} C_DIS
LIN {X -7.3899,Y 1.5627,Z 9,A -3.0071,B 0,C 0,E1 0.1598,E2 90.0712} C_DIS
LIN {X -7.5203,Y 0.6934,Z 9,A -3.0485,B 0,C 0,E1 0.1598,E2 90.0712} C_DIS
LIN {X -7.5423,Y -0.4711,Z 9,A -3.0981,B 0,C 0,E1 0.1598,E2 90.0708} C_DIS
LIN {X -7.3701,Y -1.6545,Z 9,A -3.1415,B 0,C 0,E1 0.1598,E2 90.0707} C_DIS
LIN {X -7.0937,Y -2.6041,Z 9,A -3.1715,B 0,C 0,E1 0.1598,E2 90.0707} C_DIS
LIN {X -6.6436,Y -3.6006,Z 9,A -3.197,B 0,C 0,E1 0.1598,E2 90.0708} C_DIS
LIN {X -5.918,Y -4.6999,Z 9,A -3.2166,B 0,C 0,E1 0.1598,E2 90.0707} C_DIS
LIN {X -5.195,Y -5.4873,Z 9,A -3.2235,B 0,C 0,E1 0.1598,E2 90.0709} C_DIS
LIN {X -4.3984,Y -6.1402,Z 9,A -3.222,B 0,C 0,E1 0.1598,E2 90.0711} C_DIS
LIN {X -3.7034,Y -6.5829,Z 9,A -3.2153,B 0,C 0,E1 0.1598,E2 90.0711} C_DIS
LIN {X -2.6579,Y -7.0739,Z 9,A -3.1977,B 0,C 0,E1 0.1598,E2 90.0711} C_DIS
LIN {X -1.7146,Y -7.3615,Z 9,A -3.1753,B 0,C 0,E1 0.1598,E2 90.0713} C_DIS
LIN {X -0.8195,Y -7.5124,Z 9,A -3.1489,B 0,C 0,E1 0.1598,E2 90.0713} C_DIS
LIN {X -0.0391,Y -7.5523,Z 9,A -3.122,B 0,C 0,E1 0.1598,E2 90.0714} C_DIS
Enddeposition()
LIN {X -0.0391,Y -7.5523,Z 9,A -3.122,B 0,C 0,E1 0.1598,E2 90.0714} C_DIS
Startdeposition()
$VEL.CP = VEL_PRINT
LIN {X -0.6658,Y -8.4621,Z 9,A -3.1831,B 0,C 0,E1 0.1598,E2 90.0708} C_DIS
LIN {X -1.6629,Y -8.3263,Z 9,A -3.2145,B 0,C 0,E1 0.1598,E2 90.0712} C_DIS
LIN {X -2.7649,Y -8.0231,Z 9,A -3.242,B 0,C 0,E1 0.1598,E2 90.0712} C_DIS
LIN {X -3.5203,Y -7.722,Z 9,A -3.257,B 0,C 0,E1 0.1598,E2 90.0712} C_DIS
LIN {X -4.2436,Y -7.35,Z 9,A -3.2678,B 0,C 0,E1 0.1598,E2 90.0712} C_DIS
LIN {X -4.9281,Y -6.9107,Z 9,A -3.2743,B 0,C 0,E1 0.1598,E2 90.0712} C_DIS
LIN {X -5.5675,Y -6.408,Z 9,A -3.2765,B 0,C 0,E1 0.1598,E2 90.0711} C_DIS
LIN {X -6.296,Y -5.6989,Z 9,A -3.2731,B 0,C 0,E1 0.1598,E2 90.0709} C_DIS
LIN {X -7.0132,Y -4.7818,Z 9,A -3.2606,B 0,C 0,E1 0.1598,E2 90.0708} C_DIS
LIN {X -7.5952,Y -3.7953,Z 9,A -3.2403,B 0,C 0,E1 0.1598,E2 90.0708} C_DIS
LIN {X -8.0753,Y -2.6235,Z 9,A -3.2084,B 0,C 0,E1 0.1598,E2 90.0706} C_DIS
LIN {X -8.364,Y -1.4446,Z 9,A -3.1693,B 0,C 0,E1 0.1598,E2 90.0706} C_DIS
LIN {X -8.4665,Y -0.6423,Z 9,A -3.1396,B 0,C 0,E1 0.1598,E2 90.0709} C_DIS
LIN {X -8.4785,Y 0.3779,Z 9,A -3.0971,B 0,C 0,E1 0.1598,E2 90.0709} C_DIS
LIN {X -8.4022,Y 1.1906,Z 9,A -3.0603,B 0,C 0,E1 0.1598,E2 90.0712} C_DIS
LIN {X -8.2488,Y 1.9924,Z 9,A -3.0209,B 0,C 0,E1 0.1598,E2 90.0712} C_DIS
LIN {X -8.0193,Y 2.7758,Z 9,A -2.9795,B 0,C 0,E1 0.1598,E2 90.0712} C_DIS
LIN {X -7.7157,Y 3.5336,Z 9,A -2.9365,B 0,C 0,E1 0.1598,E2 90.0714} C_DIS
LIN {X -7.3408,Y 4.2588,Z 9,A -2.8922,B 0,C 0,E1 0.1598,E2 90.0714} C_DIS
LIN {X -6.8982,Y 4.9449,Z 9,A -2.8471,B 0,C 0,E1 0.1598,E2 90.0715} C_DIS
LIN {X -6.392,Y 5.5854,Z 9,A -2.8015,B 0,C 0,E1 0.1598,E2 90.0716} C_DIS
LIN {X -5.8265,Y 6.1744,Z 9,A -2.7559,B 0,C 0,E1 0.1598,E2 90.0717} C_DIS
LIN {X -5.2063,Y 6.7054,Z 9,A -2.7107,B 0,C 0,E1 0.1598,E2 90.0718} C_DIS
LIN {X -4.5376,Y 7.1738,Z 9,A -2.6663,B 0,C 0,E1 0.1598,E2 90.0719} C_DIS
LIN {X -3.827,Y 7.5758,Z 9,A -2.6232,B 0,C 0,E1 0.1598,E2 90.0719} C_DIS
LIN {X -3.0813,Y 7.908,Z 9,A -2.5817,B 0,C 0,E1 0.1598,E2 90.0721} C_DIS
LIN {X -2.3072,Y 8.1673,Z 9,A -2.5422,B 0,C 0,E1 0.1598,E2 90.0721} C_DIS
LIN {X -1.1845,Y 8.409,Z 9,A -2.4906,B 0,C 0,E1 0.1598,E2 90.0722} C_DIS
LIN {X -0.1456,Y 8.4874,Z 9,A -2.4489,B 0,C 0,E1 0.1598,E2 90.0723} C_DIS
LIN {X 0.6874,Y 8.4598,Z 9,A -2.4193,B 0,C 0,E1 0.1598,E2 90.0723} C_DIS
LIN {X 1.5137,Y 8.3509,Z 9,A -2.3934,B 0,C 0,E1 0.1598,E2 90.0723} C_DIS
LIN {X 2.3255,Y 8.1622,Z 9,A -2.3713,B 0,C 0,E1 0.1598,E2 90.0723} C_DIS
LIN {X 3.1149,Y 7.8947,Z 9,A -2.3535,B 0,C 0,E1 0.1598,E2 90.0723} C_DIS
LIN {X 3.8743,Y 7.5511,Z 9,A -2.3399,B 0,C 0,E1 0.1598,E2 90.0723} C_DIS
LIN {X 4.5965,Y 7.135,Z 9,A -2.3308,B 0,C 0,E1 0.1598,E2 90.0723} C_DIS
LIN {X 5.2744,Y 6.65,Z 9,A -2.3263,B 0,C 0,E1 0.1598,E2 90.0723} C_DIS
LIN {X 5.9017,Y 6.1012,Z 9,A -2.3263,B 0,C 0,E1 0.1598,E2 90.0723} C_DIS
LIN {X 6.4718,Y 5.4932,Z 9,A -2.331,B 0,C 0,E1 0.1598,E2 90.0723} C_DIS
LIN {X 6.9791,Y 4.8319,Z 9,A -2.3403,B 0,C 0,E1 0.1598,E2 90.0722} C_DIS
LIN {X 7.419,Y 4.1239,Z 9,A -2.3541,B 0,C 0,E1 0.1598,E2 90.0722} C_DIS
LIN {X 7.7875,Y 3.3763,Z 9,A -2.3722,B 0,C 0,E1 0.1598,E2 90.0721} C_DIS
LIN {X 8.0813,Y 2.5963,Z 9,A -2.3944,B 0,C 0,E1 0.1598,E2 90.0721} C_DIS
LIN {X 8.3654,Y 1.4554,Z 9,A -2.432,B 0,C 0,E1 0.1598,E2 90.0716} C_DIS
LIN {X 8.4905,Y 0.0954,Z 9,A -2.4848,B 0,C 0,E1 0.1598,E2 90.0712} C_DIS
LIN {X 8.418,Y -1.0833,Z 9,A -2.5378,B 0,C 0,E1 0.1598,E2 90.0714} C_DIS
LIN {X 8.2743,Y -1.8892,Z 9,A -2.5777,B 0,C 0,E1 0.1598,E2 90.0718} C_DIS
LIN {X 8.0539,Y -2.6776,Z 9,A -2.6193,B 0,C 0,E1 0.1598,E2 90.0718} C_DIS
LIN {X 7.7588,Y -3.4413,Z 9,A -2.6627,B 0,C 0,E1 0.1598,E2 90.0718} C_DIS
LIN {X 7.2423,Y -4.4307,Z 9,A -2.7235,B 0,C 0,E1 0.1598,E2 90.0715} C_DIS
LIN {X 6.6482,Y -5.2766,Z 9,A -2.7814,B 0,C 0,E1 0.1598,E2 90.0715} C_DIS
LIN {X 6.1038,Y -5.8992,Z 9,A -2.8279,B 0,C 0,E1 0.1598,E2 90.0716} C_DIS
LIN {X 5.5013,Y -6.4656,Z 9,A -2.8741,B 0,C 0,E1 0.1598,E2 90.0716} C_DIS
LIN {X 4.6762,Y -7.0885,Z 9,A -2.9308,B 0,C 0,E1 0.1598,E2 90.0715} C_DIS
LIN {X 3.9249,Y -7.5306,Z 9,A -2.9772,B 0,C 0,E1 0.1598,E2 90.0715} C_DIS
LIN {X 2.9083,Y -7.9738,Z 9,A -3.0333,B 0,C 0,E1 0.1598,E2 90.0715} C_DIS
LIN {X 2.2292,Y -8.1909,Z 9,A -3.0675,B 0,C 0,E1 0.1598,E2 90.0715} C_DIS
LIN {X 1.5336,Y -8.3479,Z 9,A -3.0996,B 0,C 0,E1 0.1598,E2 90.0715} C_DIS
LIN {X 0.8276,Y -8.4476,Z 9,A -3.1297,B 0,C 0,E1 0.1598,E2 90.0715} C_DIS
LIN {X -0.0625,Y -8.4906,Z 9,A -3.1642,B 0,C 0,E1 0.1598,E2 90.0714} C_DIS
Enddeposition()
LIN {X 0.0003,Y -4.7568,Z 10,A -2.9885,B 0,C 0,E1 0.1598,E2 90.0604} C_DIS
Startdeposition()
$VEL.CP = VEL_PRINT
LIN {X 0.0003,Y -4.7568,Z 10,A -2.9941,B 0,C 0,E1 0.1598,E2 90.0661} C_DIS
LIN {X 0.8439,Y -4.6766,Z 10,A -2.9646,B 0,C 0,E1 0.1598,E2 90.071} C_DIS
LIN {X 1.5007,Y -4.5083,Z 10,A -2.934,B 0,C 0,E1 0.1598,E2 90.0716} C_DIS
LIN {X 2.127,Y -4.2487,Z 10,A -2.9,B 0,C 0,E1 0.1598,E2 90.0716} C_DIS
LIN {X 2.7087,Y -3.9007,Z 10,A -2.8638,B 0,C 0,E1 0.1598,E2 90.0716} C_DIS
LIN {X 3.2379,Y -3.4771,Z 10,A -2.8264,B 0,C 0,E1 0.1598,E2 90.0717} C_DIS
LIN {X 3.7002,Y -2.9813,Z 10,A -2.7884,B 0,C 0,E1 0.1598,E2 90.0717} C_DIS
LIN {X 4.0875,Y -2.4248,Z 10,A -2.7505,B 0,C 0,E1 0.1598,E2 90.0717} C_DIS
LIN {X 4.3891,Y -1.8177,Z 10,A -2.7136,B 0,C 0,E1 0.1598,E2 90.0717} C_DIS
LIN {X 4.6033,Y -1.1746,Z 10,A -2.6785,B 0,C 0,E1 0.1598,E2 90.0717} C_DIS
LIN {X 4.7239,Y -0.5076,Z 10,A -2.6457,B 0,C 0,E1 0.1598,E2 90.0718} C_DIS
LIN {X 4.7491,Y 0.1699,Z 10,A -2.6161,B 0,C 0,E1 0.1598,E2 90.0718} C_DIS
LIN {X 4.6758,Y 0.8438,Z 10,A -2.5902,B 0,C 0,E1 0.1598,E2 90.0718} C_DIS
LIN {X 4.5077,Y 1.5006,Z 10,A -2.5686,B 0,C 0,E1 0.1598,E2 90.0719} C_DIS
LIN {X 4.2491,Y 2.1272,Z 10,A -2.5516,B 0,C 0,E1 0.1598,E2 90.0719} C_DIS
LIN {X 3.9035,Y 2.7105,Z 10,A -2.5396,B 0,C 0,E1 0.1598,E2 90.0719} C_DIS
LIN {X 3.477,Y 3.2375,Z 10,A -2.5331,B 0,C 0,E1 0.1598,E2 90.072} C_DIS
LIN {X 2.9812,Y 3.6997,Z 10,A -2.5318,B 0,C 0,E1 0.1598,E2 90.072} C_DIS
LIN {X 2.4239,Y 4.0859,Z 10,A -2.5361,B 0,C 0,E1 0.1598,E2 90.0721} C_DIS
LIN {X 1.8173,Y 4.3882,Z 10,A -2.5457,B 0,C 0,E1 0.1598,E2 90.0721} C_DIS
LIN {X 1.1744,Y 4.6025,Z 10,A -2.5603,B 0,C 0,E1 0.1598,E2 90.0721} C_DIS
LIN {X 0.5076,Y 4.7238,Z 10,A -2.5798,B 0,C 0,E1 0.1598,E2 90.0721} C_DIS
LIN {X -0.1699,Y 4.7493,Z 10,A -2.6037,B 0,C 0,E1 0.1598,E2 90.0721} C_DIS
LIN {X -0.8438,Y 4.6759,Z 10,A -2.6317,B 0,C 0,E1 0.1598,E2 90.0721} C_DIS
LIN {X -1.5006,Y 4.5079,Z 10,A -2.663,B 0,C 0,E1 0.1598,E2 90.0721} C_DIS
LIN {X -2.1275,Y 4.2497,Z 10,A -2.697,B 0,C 0,E1 0.1598,E2 90.0719} C_DIS
LIN {X -2.7103,Y 3.9031,Z 10,A -2.733,B 0,C 0,E1 0.1598,E2 90.0719} C_DIS
LIN {X -3.2383,Y 3.4778,Z 10,A -2.7704,B 0,C 0,E1 0.1598,E2 90.0718} C_DIS
LIN {X -3.7,Y 2.9815,Z 10,A -2.8083,B 0,C 0,E1 0.1598,E2 90.0718} C_DIS
LIN {X -4.087,Y 2.4247,Z 10,A -2.846,B 0,C 0,E1 0.1598,E2 90.0716} C_DIS
LIN {X -4.3886,Y 1.8177,Z 10,A -2.8826,B 0,C 0,E1 0.1598,E2 90.0716} C_DIS
LIN {X -4.6022,Y 1.1745,Z 10,A -2.9176,B 0,C 0,E1 0.1598,E2 90.0715} C_DIS
LIN {X -4.7244,Y 0.5076,Z 10,A -2.9502,B 0,C 0,E1 0.1598,E2 90.0715} C_DIS
LIN {X -4.7469,Y -0.1698,Z 10,A -2.9796,B 0,C 0,E1 0.1598,E2 90.0714} C_DIS
LIN {X -4.676,Y -0.8439,Z 10,A -3.0054,B 0,C 0,E1 0.1598,E2 90.0714} C_DIS
LIN {X -4.5084,Y -1.5008,Z 10,A -3.0269,B 0,C 0,E1 0.1598,E2 90.0714} C_DIS
LIN {X -4.2488,Y -2.127,Z 10,A -3.0438,B 0,C 0,E1 0.1598,E2 90.0714} C_DIS
LIN {X -3.9026,Y -2.71,Z 10,A -3.0557,B 0,C 0,E1 0.1598,E2 90.0714} C_DIS
LIN {X -3.4756,Y -3.2363,Z 10,A -3.0623,B 0,C 0,E1 0.1598,E2 90.0714} C_DIS
LIN {X -2.9813,Y -3.7003,Z 10,A -3.0638,B 0,C 0,E1 0.1598,E2 90.0714} C_DIS
LIN {X -2.4246,Y -4.0873,Z 10,A -3.0597,B 0,C 0,E1 0.1598,E2 90.0714} C_DIS
LIN {X -1.8175,Y -4.3888,Z 10,A -3.0502,B 0,C 0,E1 0.1598,E2 90.0714} C_DIS
LIN {X -1.1745,Y -4.603,Z 10,A -3.0357,B 0,C 0,E1 0.1598,E2 90.0715} C_DIS
LIN {X -0.5075,Y -4.7246,Z 10,A -3.0163,B 0,C 0,E1 0.1598,E2 90.0715} C_DIS
LIN {X -0.5075,Y -4.7246,Z 10,A -3.0163,B 0,C 0,E1 0.1598,E2 90.0715} C_DIS
Enddeposition()
LIN {X -0.0074,Y -5.6863,Z 10,A -3.0377,B 0,C 0,E1 0.1598,E2 90.0704} C_DIS
Startdeposition()
$VEL.CP = VEL_PRINT
LIN {X -0.9748,Y -5.6002,Z 10,A -3.0706,B 0,C 0,E1 0.1598,E2 90.0714} C_DIS
LIN {X -1.7303,Y -5.4169,Z 10,A -3.0906,B 0,C 0,E1 0.1598,E2 90.0714} C_DIS
LIN {X -2.4522,Y -5.1286,Z 10,A -3.1049,B 0,C 0,E1 0.1598,E2 90.0714} C_DIS
LIN {X -3.1295,Y -4.747,Z 10,A -3.1136,B 0,C 0,E1 0.1598,E2 90.0714} C_DIS
LIN {X -3.7456,Y -4.2733,Z 10,A -3.1162,B 0,C 0,E1 0.1598,E2 90.0713} C_DIS
LIN {X -4.2941,Y -3.7229,Z 10,A -3.113,B 0,C 0,E1 0.1598,E2 90.0713} C_DIS
LIN {X -4.7617,Y -3.1022,Z 10,A -3.104,B 0,C 0,E1 0.1598,E2 90.0713} C_DIS
LIN {X -5.1413,Y -2.424,Z 10,A -3.0893,B 0,C 0,E1 0.1598,E2 90.0713} C_DIS
LIN {X -5.4244,Y -1.7002,Z 10,A -3.0691,B 0,C 0,E1 0.1598,E2 90.0713} C_DIS
LIN {X -5.6045,Y -0.9441,Z 10,A -3.0438,B 0,C 0,E1 0.1598,E2 90.0713} C_DIS
LIN {X -5.6804,Y -0.1707,Z 10,A -3.014,B 0,C 0,E1 0.1598,E2 90.0713} C_DIS
LIN {X -5.6508,Y 0.6057,Z 10,A -2.9802,B 0,C 0,E1 0.1598,E2 90.0713} C_DIS
LIN {X -5.5156,Y 1.3709,Z 10,A -2.943,B 0,C 0,E1 0.1598,E2 90.0713} C_DIS
LIN {X -5.1578,Y 2.4027,Z 10,A -2.8861,B 0,C 0,E1 0.1598,E2 90.0713} C_DIS
LIN {X -4.6987,Y 3.2004,Z 10,A -2.8358,B 0,C 0,E1 0.1598,E2 90.0715} C_DIS
LIN {X -4.2444,Y 3.7798,Z 10,A -2.7948,B 0,C 0,E1 0.1598,E2 90.0717} C_DIS
LIN {X -3.7205,Y 4.2967,Z 10,A -2.7537,B 0,C 0,E1 0.1598,E2 90.0717} C_DIS
LIN {X -2.6712,Y 5.0238,Z 10,A -2.6843,B 0,C 0,E1 0.1598,E2 90.0717} C_DIS
LIN {X -1.5178,Y 5.4777,Z 10,A -2.6227,B 0,C 0,E1 0.1598,E2 90.072} C_DIS
LIN {X -0.7178,Y 5.6398,Z 10,A -2.5865,B 0,C 0,E1 0.1598,E2 90.0721} C_DIS
LIN {X 0.0973,Y 5.6853,Z 10,A -2.5545,B 0,C 0,E1 0.1598,E2 90.0721} C_DIS
LIN {X 0.9103,Y 5.6118,Z 10,A -2.5276,B 0,C 0,E1 0.1598,E2 90.0721} C_DIS
LIN {X 1.7046,Y 5.4234,Z 10,A -2.5062,B 0,C 0,E1 0.1598,E2 90.0722} C_DIS
LIN {X 2.4636,Y 5.123,Z 10,A -2.4909,B 0,C 0,E1 0.1598,E2 90.0722} C_DIS
LIN {X 3.1714,Y 4.7165,Z 10,A -2.482,B 0,C 0,E1 0.1598,E2 90.0722} C_DIS
LIN {X 3.8137,Y 4.213,Z 10,A -2.4795,B 0,C 0,E1 0.1598,E2 90.0722} C_DIS
LIN {X 4.3774,Y 3.6229,Z 10,A -2.4837,B 0,C 0,E1 0.1598,E2 90.0721} C_DIS
LIN {X 4.8525,Y 2.9595,Z 10,A -2.4942,B 0,C 0,E1 0.1598,E2 90.072} C_DIS
LIN {X 5.2261,Y 2.2338,Z 10,A -2.5112,B 0,C 0,E1 0.1598,E2 90.072} C_DIS
LIN {X 5.4928,Y 1.4626,Z 10,A -2.534,B 0,C 0,E1 0.1598,E2 90.0719} C_DIS
LIN {X 5.6465,Y 0.661,Z 10,A -2.5623,B 0,C 0,E1 0.1598,E2 90.0718} C_DIS
LIN {X 5.6826,Y -0.1545,Z 10,A -2.5955,B 0,C 0,E1 0.1598,E2 90.0718} C_DIS
LIN {X 5.601,Y -0.9666,Z 10,A -2.633,B 0,C 0,E1 0.1598,E2 90.0718} C_DIS
LIN {X 5.4051,Y -1.7589,Z 10,A -2.6738,B 0,C 0,E1 0.1598,E2 90.0717} C_DIS
LIN {X 5.096,Y -2.5142,Z 10,A -2.7173,B 0,C 0,E1 0.1598,E2 90.0717} C_DIS
LIN {X 4.686,Y -3.2198,Z 10,A -2.7623,B 0,C 0,E1 0.1598,E2 90.0717} C_DIS
LIN {X 4.1747,Y -3.8561,Z 10,A -2.8081,B 0,C 0,E1 0.1598,E2 90.0717} C_DIS
LIN {X 3.579,Y -4.4138,Z 10,A -2.8537,B 0,C 0,E1 0.1598,E2 90.0717} C_DIS
LIN {X 2.9101,Y -4.8813,Z 10,A -2.8981,B 0,C 0,E1 0.1598,E2 90.0717} C_DIS
LIN {X 2.181,Y -5.2476,Z 10,A -2.9405,B 0,C 0,E1 0.1598,E2 90.0716} C_DIS
LIN {X 1.407,Y -5.5061,Z 10,A -2.9798,B 0,C 0,E1 0.1598,E2 90.0716} C_DIS
LIN {X 0.6039,Y -5.6497,Z 10,A -3.0154,B 0,C 0,E1 0.1598,E2 90.0716} C_DIS
LIN {X 0.6039,Y -5.6497,Z 10,A -3.0154,B 0,C 0,E1 0.1598,E2 90.0716} C_DIS
Enddeposition()
LIN {X -0.0261,Y -6.6197,Z 10,A -3.0786,B 0,C 0,E1 0.1598,E2 90.0703} C_DIS
Startdeposition()
$VEL.CP = VEL_PRINT
LIN {X 0.995,Y -6.5483,Z 10,A -3.0392,B 0,C 0,E1 0.1598,E2 90.0715} C_DIS
LIN {X 1.8298,Y -6.3613,Z 10,A -3.0007,B 0,C 0,E1 0.1598,E2 90.0715} C_DIS
LIN {X 2.477,Y -6.1383,Z 10,A -2.9675,B 0,C 0,E1 0.1598,E2 90.0715} C_DIS
LIN {X 3.0984,Y -5.8512,Z 10,A -2.9325,B 0,C 0,E1 0.1598,E2 90.0716} C_DIS
LIN {X 3.6845,Y -5.4977,Z 10,A -2.896,B 0,C 0,E1 0.1598,E2 90.0716} C_DIS
LIN {X 4.2329,Y -5.0882,Z 10,A -2.8585,B 0,C 0,E1 0.1598,E2 90.0716} C_DIS
LIN {X 4.7357,Y -4.6238,Z 10,A -2.8203,B 0,C 0,E1 0.1598,E2 90.0717} C_DIS
LIN {X 5.1882,Y -4.1102,Z 10,A -2.7818,B 0,C 0,E1 0.1598,E2 90.0717} C_DIS
LIN {X 5.5865,Y -3.5534,Z 10,A -2.7436,B 0,C 0,E1 0.1598,E2 90.0717} C_DIS
LIN {X 5.9239,Y -2.9579,Z 10,A -2.7059,B 0,C 0,E1 0.1598,E2 90.0717} C_DIS
LIN {X 6.197,Y -2.3302,Z 10,A -2.6691,B 0,C 0,E1 0.1598,E2 90.0718} C_DIS
LIN {X 6.4042,Y -1.6778,Z 10,A -2.6338,B 0,C 0,E1 0.1598,E2 90.0718} C_DIS
LIN {X 6.541,Y -1.0071,Z 10,A -2.6003,B 0,C 0,E1 0.1598,E2 90.0718} C_DIS
LIN {X 6.6122,Y -0.3265,Z 10,A -2.5688,B 0,C 0,E1 0.1598,E2 90.0718} C_DIS
LIN {X 6.5876,Y 0.6884,Z 10,A -2.5263,B 0,C 0,E1 0.1598,E2 90.0717} C_DIS
LIN {X 6.4009,Y 1.6874,Z 10,A -2.4909,B 0,C 0,E1 0.1598,E2 90.0717} C_DIS
LIN {X 6.1443,Y 2.459,Z 10,A -2.4677,B 0,C 0,E1 0.1598,E2 90.0719} C_DIS
LIN {X 5.7977,Y 3.1945,Z 10,A -2.4494,B 0,C 0,E1 0.1598,E2 90.0719} C_DIS
LIN {X 5.362,Y 3.881,Z 10,A -2.4364,B 0,C 0,E1 0.1598,E2 90.072} C_DIS
LIN {X 4.639,Y 4.7278,Z 10,A -2.427,B 0,C 0,E1 0.1598,E2 90.072} C_DIS
LIN {X 3.953,Y 5.3092,Z 10,A -2.4279,B 0,C 0,E1 0.1598,E2 90.0721} C_DIS
LIN {X 3.3537,Y 5.7069,Z 10,A -2.4333,B 0,C 0,E1 0.1598,E2 90.0722} C_DIS
LIN {X 2.714,Y 6.0356,Z 10,A -2.443,B 0,C 0,E1 0.1598,E2 90.0722} C_DIS
LIN {X 2.0435,Y 6.2959,Z 10,A -2.4568,B 0,C 0,E1 0.1598,E2 90.0722} C_DIS
LIN {X 1.3485,Y 6.481,Z 10,A -2.4746,B 0,C 0,E1 0.1598,E2 90.0722} C_DIS
LIN {X 0.6372,Y 6.5873,Z 10,A -2.4964,B 0,C 0,E1 0.1598,E2 90.0722} C_DIS
LIN {X -0.0813,Y 6.6192,Z 10,A -2.5216,B 0,C 0,E1 0.1598,E2 90.0722} C_DIS
LIN {X -0.7988,Y 6.5696,Z 10,A -2.5502,B 0,C 0,E1 0.1598,E2 90.0722} C_DIS
LIN {X -1.5074,Y 6.4468,Z 10,A -2.5815,B 0,C 0,E1 0.1598,E2 90.0722} C_DIS
LIN {X -2.1979,Y 6.2455,Z 10,A -2.6154,B 0,C 0,E1 0.1598,E2 90.0721} C_DIS
LIN {X -2.8628,Y 5.971,Z 10,A -2.6515,B 0,C 0,E1 0.1598,E2 90.0721} C_DIS
LIN {X -3.4917,Y 5.6218,Z 10,A -2.6894,B 0,C 0,E1 0.1598,E2 90.0719} C_DIS
LIN {X -4.0824,Y 5.2115,Z 10,A -2.7285,B 0,C 0,E1 0.1598,E2 90.0719} C_DIS
LIN {X -4.6236,Y 4.738,Z 10,A -2.7683,B 0,C 0,E1 0.1598,E2 90.0718} C_DIS
LIN {X -5.11,Y 4.208,Z 10,A -2.8086,B 0,C 0,E1 0.1598,E2 90.0717} C_DIS
LIN {X -5.537,Y 3.6292,Z 10,A -2.8486,B 0,C 0,E1 0.1598,E2 90.0717} C_DIS
LIN {X -5.8982,Y 3.0072,Z 10,A -2.8881,B 0,C 0,E1 0.1598,E2 90.0715} C_DIS
LIN {X -6.1892,Y 2.3495,Z 10,A -2.9265,B 0,C 0,E1 0.1598,E2 90.0715} C_DIS
LIN {X -6.4078,Y 1.6642,Z 10,A -2.9634,B 0,C 0,E1 0.1598,E2 90.0714} C_DIS
LIN {X -6.5506,Y 0.9593,Z 10,A -2.9983,B 0,C 0,E1 0.1598,E2 90.0714} C_DIS
LIN {X -6.6149,Y 0.2428,Z 10,A -3.0308,B 0,C 0,E1 0.1598,E2 90.0713} C_DIS
LIN {X -6.6011,Y -0.4763,Z 10,A -3.0606,B 0,C 0,E1 0.1598,E2 90.0713} C_DIS
LIN {X -6.5118,Y -1.1898,Z 10,A -3.0874,B 0,C 0,E1 0.1598,E2 90.0712} C_DIS
LIN {X -6.3432,Y -1.8891,Z 10,A -3.1106,B 0,C 0,E1 0.1598,E2 90.0712} C_DIS
LIN {X -6.1026,Y -2.5669,Z 10,A -3.1304,B 0,C 0,E1 0.1598,E2 90.0712} C_DIS
LIN {X -5.7863,Y -3.2129,Z 10,A -3.146,B 0,C 0,E1 0.1598,E2 90.0712} C_DIS
LIN {X -5.4056,Y -3.8232,Z 10,A -3.1578,B 0,C 0,E1 0.1598,E2 90.0712} C_DIS
LIN {X -4.9579,Y -4.3863,Z 10,A -3.1651,B 0,C 0,E1 0.1598,E2 90.0712} C_DIS
LIN {X -4.4525,Y -4.8982,Z 10,A -3.1682,B 0,C 0,E1 0.1598,E2 90.0712} C_DIS
LIN {X -3.8949,Y -5.3525,Z 10,A -3.167,B 0,C 0,E1 0.1598,E2 90.0712} C_DIS
LIN {X -3.2907,Y -5.7425,Z 10,A -3.1613,B 0,C 0,E1 0.1598,E2 90.0712} C_DIS
LIN {X -2.6481,Y -6.0657,Z 10,A -3.1514,B 0,C 0,E1 0.1598,E2 90.0713} C_DIS
LIN {X -1.9743,Y -6.317,Z 10,A -3.1373,B 0,C 0,E1 0.1598,E2 90.0713} C_DIS
LIN {X -1.2773,Y -6.4942,Z 10,A -3.1193,B 0,C 0,E1 0.1598,E2 90.0713} C_DIS
LIN {X -0.5653,Y -6.5964,Z 10,A -3.0975,B 0,C 0,E1 0.1598,E2 90.0714} C_DIS
LIN {X -0.5653,Y -6.5964,Z 10,A -3.0975,B 0,C 0,E1 0.1598,E2 90.0714} C_DIS
Enddeposition()
LIN {X -0.0044,Y -7.5545,Z 10,A -3.1165,B 0,C 0,E1 0.1598,E2 90.0703} C_DIS
Startdeposition()
$VEL.CP = VEL_PRINT
LIN {X -0.8594,Y -7.5078,Z 10,A -3.147,B 0,C 0,E1 0.1598,E2 90.0713} C_DIS
LIN {X -1.8815,Y -7.3187,Z 10,A -3.1765,B 0,C 0,E1 0.1598,E2 90.0713} C_DIS
LIN {X -2.8192,Y -7.0078,Z 10,A -3.1977,B 0,C 0,E1 0.1598,E2 90.0713} C_DIS
LIN {X -3.5359,Y -6.6747,Z 10,A -3.2099,B 0,C 0,E1 0.1598,E2 90.0713} C_DIS
LIN {X -4.2138,Y -6.2685,Z 10,A -3.2176,B 0,C 0,E1 0.1598,E2 90.0712} C_DIS
LIN {X -4.8453,Y -5.7933,Z 10,A -3.2207,B 0,C 0,E1 0.1598,E2 90.0712} C_DIS
LIN {X -5.5634,Y -5.1149,Z 10,A -3.2182,B 0,C 0,E1 0.1598,E2 90.071} C_DIS
LIN {X -6.2463,Y -4.2527,Z 10,A -3.2068,B 0,C 0,E1 0.1598,E2 90.0709} C_DIS
LIN {X -6.793,Y -3.31,Z 10,A -3.187,B 0,C 0,E1 0.1598,E2 90.0709} C_DIS
LIN {X -7.1932,Y -2.3162,Z 10,A -3.1598,B 0,C 0,E1 0.1598,E2 90.0709} C_DIS
LIN {X -7.4312,Y -1.3514,Z 10,A -3.128,B 0,C 0,E1 0.1598,E2 90.0709} C_DIS
LIN {X -7.5538,Y -0.2259,Z 10,A -3.0849,B 0,C 0,E1 0.1598,E2 90.0709} C_DIS
LIN {X -7.4907,Y 0.968,Z 10,A -3.0322,B 0,C 0,E1 0.1598,E2 90.0708} C_DIS
LIN {X -7.2766,Y 2.0433,Z 10,A -2.9791,B 0,C 0,E1 0.1598,E2 90.0709} C_DIS
LIN {X -6.8802,Y 3.1162,Z 10,A -2.9195,B 0,C 0,E1 0.1598,E2 90.0711} C_DIS
LIN {X -6.518,Y 3.8156,Z 10,A -2.877,B 0,C 0,E1 0.1598,E2 90.0715} C_DIS
LIN {X -6.0857,Y 4.4741,Z 10,A -2.8334,B 0,C 0,E1 0.1598,E2 90.0715} C_DIS
LIN {X -5.5865,Y 5.0835,Z 10,A -2.7894,B 0,C 0,E1 0.1598,E2 90.0717} C_DIS
LIN {X -4.8801,Y 5.7694,Z 10,A -2.7344,B 0,C 0,E1 0.1598,E2 90.0717} C_DIS
LIN {X -3.968,Y 6.4263,Z 10,A -2.6731,B 0,C 0,E1 0.1598,E2 90.0717} C_DIS
LIN {X -3.2649,Y 6.8092,Z 10,A -2.6312,B 0,C 0,E1 0.1598,E2 90.072} C_DIS
LIN {X -2.5267,Y 7.1188,Z 10,A -2.5909,B 0,C 0,E1 0.1598,E2 90.072} C_DIS
LIN {X -1.7588,Y 7.3461,Z 10,A -2.553,B 0,C 0,E1 0.1598,E2 90.0721} C_DIS
LIN {X -0.7727,Y 7.5177,Z 10,A -2.5094,B 0,C 0,E1 0.1598,E2 90.0722} C_DIS
LIN {X 0.2361,Y 7.5536,Z 10,A -2.4706,B 0,C 0,E1 0.1598,E2 90.0722} C_DIS
LIN {X 1.454,Y 7.4123,Z 10,A -2.4316,B 0,C 0,E1 0.1598,E2 90.0723} C_DIS
LIN {X 2.1991,Y 7.2298,Z 10,A -2.4118,B 0,C 0,E1 0.1598,E2 90.0723} C_DIS
LIN {X 3.1313,Y 6.8795,Z 10,A -2.3921,B 0,C 0,E1 0.1598,E2 90.0723} C_DIS
LIN {X 4.2595,Y 6.2416,Z 10,A -2.3773,B 0,C 0,E1 0.1598,E2 90.0722} C_DIS
LIN {X 5.0475,Y 5.6183,Z 10,A -2.3747,B 0,C 0,E1 0.1598,E2 90.0722} C_DIS
LIN {X 5.6164,Y 5.0504,Z 10,A -2.3777,B 0,C 0,E1 0.1598,E2 90.0722} C_DIS
LIN {X 6.1217,Y 4.4253,Z 10,A -2.3856,B 0,C 0,E1 0.1598,E2 90.0722} C_DIS
LIN {X 6.5573,Y 3.7497,Z 10,A -2.3981,B 0,C 0,E1 0.1598,E2 90.0722} C_DIS
LIN {X 6.9169,Y 3.0309,Z 10,A -2.4153,B 0,C 0,E1 0.1598,E2 90.0721} C_DIS
LIN {X 7.2987,Y 1.9583,Z 10,A -2.4464,B 0,C 0,E1 0.1598,E2 90.0717} C_DIS
LIN {X 7.4728,Y 1.1258,Z 10,A -2.4756,B 0,C 0,E1 0.1598,E2 90.0719} C_DIS
LIN {X 7.5578,Y 0.0306,Z 10,A -2.5186,B 0,C 0,E1 0.1598,E2 90.0715} C_DIS
LIN {X 7.4836,Y -1.0592,Z 10,A -2.5677,B 0,C 0,E1 0.1598,E2 90.0715} C_DIS
Enddeposition()
END
